(* Logix 5000 project; controller Kollmeyer_LiveDemo_TBENLX8IOL_TBIL vendor 1 type 14 code 176 rev 32.11; software revision 32.00 *)

TASK MainTask (continuous, watchdog 500 ms) : MainProgram
TASK SafetyTask (periodic, rate 20 ms, priority 10, watchdog 20 ms, safety) : SafetyProgram

MODULES
   Local : vendor 1 type 14 code 176 (Compact 0, rev 32.11)
      TBEN_L4_8IOL : ETHERNET-MODULE (Ethernet 192.168.1.7, rev 1.1, Output RPI 10 ms)
           TBEN_L4_8IOL:I.Data[0]   // Station Status Word
           TBEN_L4_8IOL:I.Data[0].0   // Module Diagnostics Available
           TBEN_L4_8IOL:I.Data[0].1   // INFO: ARGEE Project Running
           TBEN_L4_8IOL:I.Data[0].10   // Reserved
           TBEN_L4_8IOL:I.Data[0].11   // Reserved
           TBEN_L4_8IOL:I.Data[0].12   // Reserved
           TBEN_L4_8IOL:I.Data[0].13   // Reserved
           TBEN_L4_8IOL:I.Data[0].14   // Force Mode Enabled
           TBEN_L4_8IOL:I.Data[0].15   // Reserved
           TBEN_L4_8IOL:I.Data[0].2   // Reserved
           TBEN_L4_8IOL:I.Data[0].3   // Reserved
           TBEN_L4_8IOL:I.Data[0].4   // Reserved
           TBEN_L4_8IOL:I.Data[0].5   // Reserved
           TBEN_L4_8IOL:I.Data[0].6   // Reserved
           TBEN_L4_8IOL:I.Data[0].7   // Undervoltage Field Supply V2
           TBEN_L4_8IOL:I.Data[0].8   // Reserved
           TBEN_L4_8IOL:I.Data[0].9   // Undervoltage Field Supply V1
           TBEN_L4_8IOL:I.Data[100]   // IO-Link Port 7 - Input data word 1
           TBEN_L4_8IOL:I.Data[100].0   // IO-Link Port 7 - Input data word 1 (INT bit0)
           TBEN_L4_8IOL:I.Data[100].1   // IO-Link Port 7 - Input data word 1 (INT bit1)
           TBEN_L4_8IOL:I.Data[100].10   // IO-Link Port 7 - Input data word 1 (INT bit10)
           TBEN_L4_8IOL:I.Data[100].11   // IO-Link Port 7 - Input data word 1 (INT bit11)
           TBEN_L4_8IOL:I.Data[100].12   // IO-Link Port 7 - Input data word 1 (INT bit12)
           TBEN_L4_8IOL:I.Data[100].13   // IO-Link Port 7 - Input data word 1 (INT bit13)
           TBEN_L4_8IOL:I.Data[100].14   // IO-Link Port 7 - Input data word 1 (INT bit14)
           TBEN_L4_8IOL:I.Data[100].15   // IO-Link Port 7 - Input data word 1 (INT bit15)
           TBEN_L4_8IOL:I.Data[100].2   // IO-Link Port 7 - Input data word 1 (INT bit2)
           TBEN_L4_8IOL:I.Data[100].3   // IO-Link Port 7 - Input data word 1 (INT bit3)
           TBEN_L4_8IOL:I.Data[100].4   // IO-Link Port 7 - Input data word 1 (INT bit4)
           TBEN_L4_8IOL:I.Data[100].5   // IO-Link Port 7 - Input data word 1 (INT bit5)
           TBEN_L4_8IOL:I.Data[100].6   // IO-Link Port 7 - Input data word 1 (INT bit6)
           TBEN_L4_8IOL:I.Data[100].7   // IO-Link Port 7 - Input data word 1 (INT bit7)
           TBEN_L4_8IOL:I.Data[100].8   // IO-Link Port 7 - Input data word 1 (INT bit8)
           TBEN_L4_8IOL:I.Data[100].9   // IO-Link Port 7 - Input data word 1 (INT bit9)
           TBEN_L4_8IOL:I.Data[101]   // IO-Link Port 7 - Input data word 2
           TBEN_L4_8IOL:I.Data[101].0   // IO-Link Port 7 - Input data word 2 (INT bit0)
           TBEN_L4_8IOL:I.Data[101].1   // IO-Link Port 7 - Input data word 2 (INT bit1)
           TBEN_L4_8IOL:I.Data[101].10   // IO-Link Port 7 - Input data word 2 (INT bit10)
           TBEN_L4_8IOL:I.Data[101].11   // IO-Link Port 7 - Input data word 2 (INT bit11)
           TBEN_L4_8IOL:I.Data[101].12   // IO-Link Port 7 - Input data word 2 (INT bit12)
           TBEN_L4_8IOL:I.Data[101].13   // IO-Link Port 7 - Input data word 2 (INT bit13)
           TBEN_L4_8IOL:I.Data[101].14   // IO-Link Port 7 - Input data word 2 (INT bit14)
           TBEN_L4_8IOL:I.Data[101].15   // IO-Link Port 7 - Input data word 2 (INT bit15)
           TBEN_L4_8IOL:I.Data[101].2   // IO-Link Port 7 - Input data word 2 (INT bit2)
           TBEN_L4_8IOL:I.Data[101].3   // IO-Link Port 7 - Input data word 2 (INT bit3)
           TBEN_L4_8IOL:I.Data[101].4   // IO-Link Port 7 - Input data word 2 (INT bit4)
           TBEN_L4_8IOL:I.Data[101].5   // IO-Link Port 7 - Input data word 2 (INT bit5)
           TBEN_L4_8IOL:I.Data[101].6   // IO-Link Port 7 - Input data word 2 (INT bit6)
           TBEN_L4_8IOL:I.Data[101].7   // IO-Link Port 7 - Input data word 2 (INT bit7)
           TBEN_L4_8IOL:I.Data[101].8   // IO-Link Port 7 - Input data word 2 (INT bit8)
           TBEN_L4_8IOL:I.Data[101].9   // IO-Link Port 7 - Input data word 2 (INT bit9)
           TBEN_L4_8IOL:I.Data[102]   // IO-Link Port 7 - Input data word 3
           TBEN_L4_8IOL:I.Data[102].0   // IO-Link Port 7 - Input data word 3 (INT bit0)
           TBEN_L4_8IOL:I.Data[102].1   // IO-Link Port 7 - Input data word 3 (INT bit1)
           TBEN_L4_8IOL:I.Data[102].10   // IO-Link Port 7 - Input data word 3 (INT bit10)
           TBEN_L4_8IOL:I.Data[102].11   // IO-Link Port 7 - Input data word 3 (INT bit11)
           TBEN_L4_8IOL:I.Data[102].12   // IO-Link Port 7 - Input data word 3 (INT bit12)
           TBEN_L4_8IOL:I.Data[102].13   // IO-Link Port 7 - Input data word 3 (INT bit13)
           TBEN_L4_8IOL:I.Data[102].14   // IO-Link Port 7 - Input data word 3 (INT bit14)
           TBEN_L4_8IOL:I.Data[102].15   // IO-Link Port 7 - Input data word 3 (INT bit15)
           TBEN_L4_8IOL:I.Data[102].2   // IO-Link Port 7 - Input data word 3 (INT bit2)
           TBEN_L4_8IOL:I.Data[102].3   // IO-Link Port 7 - Input data word 3 (INT bit3)
           TBEN_L4_8IOL:I.Data[102].4   // IO-Link Port 7 - Input data word 3 (INT bit4)
           TBEN_L4_8IOL:I.Data[102].5   // IO-Link Port 7 - Input data word 3 (INT bit5)
           TBEN_L4_8IOL:I.Data[102].6   // IO-Link Port 7 - Input data word 3 (INT bit6)
           TBEN_L4_8IOL:I.Data[102].7   // IO-Link Port 7 - Input data word 3 (INT bit7)
           TBEN_L4_8IOL:I.Data[102].8   // IO-Link Port 7 - Input data word 3 (INT bit8)
           TBEN_L4_8IOL:I.Data[102].9   // IO-Link Port 7 - Input data word 3 (INT bit9)
           TBEN_L4_8IOL:I.Data[103]   // IO-Link Port 7 - Input data word 4
           TBEN_L4_8IOL:I.Data[103].0   // IO-Link Port 7 - Input data word 4 (INT bit0)
           TBEN_L4_8IOL:I.Data[103].1   // IO-Link Port 7 - Input data word 4 (INT bit1)
           TBEN_L4_8IOL:I.Data[103].10   // IO-Link Port 7 - Input data word 4 (INT bit10)
           TBEN_L4_8IOL:I.Data[103].11   // IO-Link Port 7 - Input data word 4 (INT bit11)
           TBEN_L4_8IOL:I.Data[103].12   // IO-Link Port 7 - Input data word 4 (INT bit12)
           TBEN_L4_8IOL:I.Data[103].13   // IO-Link Port 7 - Input data word 4 (INT bit13)
           TBEN_L4_8IOL:I.Data[103].14   // IO-Link Port 7 - Input data word 4 (INT bit14)
           TBEN_L4_8IOL:I.Data[103].15   // IO-Link Port 7 - Input data word 4 (INT bit15)
           TBEN_L4_8IOL:I.Data[103].2   // IO-Link Port 7 - Input data word 4 (INT bit2)
           TBEN_L4_8IOL:I.Data[103].3   // IO-Link Port 7 - Input data word 4 (INT bit3)
           TBEN_L4_8IOL:I.Data[103].4   // IO-Link Port 7 - Input data word 4 (INT bit4)
           TBEN_L4_8IOL:I.Data[103].5   // IO-Link Port 7 - Input data word 4 (INT bit5)
           TBEN_L4_8IOL:I.Data[103].6   // IO-Link Port 7 - Input data word 4 (INT bit6)
           TBEN_L4_8IOL:I.Data[103].7   // IO-Link Port 7 - Input data word 4 (INT bit7)
           TBEN_L4_8IOL:I.Data[103].8   // IO-Link Port 7 - Input data word 4 (INT bit8)
           TBEN_L4_8IOL:I.Data[103].9   // IO-Link Port 7 - Input data word 4 (INT bit9)
           TBEN_L4_8IOL:I.Data[104]   // IO-Link Port 7 - Input data word 5
           TBEN_L4_8IOL:I.Data[104].0   // IO-Link Port 7 - Input data word 5 (INT bit0)
           TBEN_L4_8IOL:I.Data[104].1   // IO-Link Port 7 - Input data word 5 (INT bit1)
           TBEN_L4_8IOL:I.Data[104].10   // IO-Link Port 7 - Input data word 5 (INT bit10)
           TBEN_L4_8IOL:I.Data[104].11   // IO-Link Port 7 - Input data word 5 (INT bit11)
           TBEN_L4_8IOL:I.Data[104].12   // IO-Link Port 7 - Input data word 5 (INT bit12)
           TBEN_L4_8IOL:I.Data[104].13   // IO-Link Port 7 - Input data word 5 (INT bit13)
           TBEN_L4_8IOL:I.Data[104].14   // IO-Link Port 7 - Input data word 5 (INT bit14)
           TBEN_L4_8IOL:I.Data[104].15   // IO-Link Port 7 - Input data word 5 (INT bit15)
           TBEN_L4_8IOL:I.Data[104].2   // IO-Link Port 7 - Input data word 5 (INT bit2)
           TBEN_L4_8IOL:I.Data[104].3   // IO-Link Port 7 - Input data word 5 (INT bit3)
           TBEN_L4_8IOL:I.Data[104].4   // IO-Link Port 7 - Input data word 5 (INT bit4)
           TBEN_L4_8IOL:I.Data[104].5   // IO-Link Port 7 - Input data word 5 (INT bit5)
           TBEN_L4_8IOL:I.Data[104].6   // IO-Link Port 7 - Input data word 5 (INT bit6)
           TBEN_L4_8IOL:I.Data[104].7   // IO-Link Port 7 - Input data word 5 (INT bit7)
           TBEN_L4_8IOL:I.Data[104].8   // IO-Link Port 7 - Input data word 5 (INT bit8)
           TBEN_L4_8IOL:I.Data[104].9   // IO-Link Port 7 - Input data word 5 (INT bit9)
           TBEN_L4_8IOL:I.Data[105]   // IO-Link Port 7 - Input data word 6
           TBEN_L4_8IOL:I.Data[105].0   // IO-Link Port 7 - Input data word 6 (INT bit0)
           TBEN_L4_8IOL:I.Data[105].1   // IO-Link Port 7 - Input data word 6 (INT bit1)
           TBEN_L4_8IOL:I.Data[105].10   // IO-Link Port 7 - Input data word 6 (INT bit10)
           TBEN_L4_8IOL:I.Data[105].11   // IO-Link Port 7 - Input data word 6 (INT bit11)
           TBEN_L4_8IOL:I.Data[105].12   // IO-Link Port 7 - Input data word 6 (INT bit12)
           TBEN_L4_8IOL:I.Data[105].13   // IO-Link Port 7 - Input data word 6 (INT bit13)
           TBEN_L4_8IOL:I.Data[105].14   // IO-Link Port 7 - Input data word 6 (INT bit14)
           TBEN_L4_8IOL:I.Data[105].15   // IO-Link Port 7 - Input data word 6 (INT bit15)
           TBEN_L4_8IOL:I.Data[105].2   // IO-Link Port 7 - Input data word 6 (INT bit2)
           TBEN_L4_8IOL:I.Data[105].3   // IO-Link Port 7 - Input data word 6 (INT bit3)
           TBEN_L4_8IOL:I.Data[105].4   // IO-Link Port 7 - Input data word 6 (INT bit4)
           TBEN_L4_8IOL:I.Data[105].5   // IO-Link Port 7 - Input data word 6 (INT bit5)
           TBEN_L4_8IOL:I.Data[105].6   // IO-Link Port 7 - Input data word 6 (INT bit6)
           TBEN_L4_8IOL:I.Data[105].7   // IO-Link Port 7 - Input data word 6 (INT bit7)
           TBEN_L4_8IOL:I.Data[105].8   // IO-Link Port 7 - Input data word 6 (INT bit8)
           TBEN_L4_8IOL:I.Data[105].9   // IO-Link Port 7 - Input data word 6 (INT bit9)
           TBEN_L4_8IOL:I.Data[106]   // IO-Link Port 7 - Input data word 7
           TBEN_L4_8IOL:I.Data[106].0   // IO-Link Port 7 - Input data word 7 (INT bit0)
           TBEN_L4_8IOL:I.Data[106].1   // IO-Link Port 7 - Input data word 7 (INT bit1)
           TBEN_L4_8IOL:I.Data[106].10   // IO-Link Port 7 - Input data word 7 (INT bit10)
           TBEN_L4_8IOL:I.Data[106].11   // IO-Link Port 7 - Input data word 7 (INT bit11)
           TBEN_L4_8IOL:I.Data[106].12   // IO-Link Port 7 - Input data word 7 (INT bit12)
           TBEN_L4_8IOL:I.Data[106].13   // IO-Link Port 7 - Input data word 7 (INT bit13)
           TBEN_L4_8IOL:I.Data[106].14   // IO-Link Port 7 - Input data word 7 (INT bit14)
           TBEN_L4_8IOL:I.Data[106].15   // IO-Link Port 7 - Input data word 7 (INT bit15)
           TBEN_L4_8IOL:I.Data[106].2   // IO-Link Port 7 - Input data word 7 (INT bit2)
           TBEN_L4_8IOL:I.Data[106].3   // IO-Link Port 7 - Input data word 7 (INT bit3)
           TBEN_L4_8IOL:I.Data[106].4   // IO-Link Port 7 - Input data word 7 (INT bit4)
           TBEN_L4_8IOL:I.Data[106].5   // IO-Link Port 7 - Input data word 7 (INT bit5)
           TBEN_L4_8IOL:I.Data[106].6   // IO-Link Port 7 - Input data word 7 (INT bit6)
           TBEN_L4_8IOL:I.Data[106].7   // IO-Link Port 7 - Input data word 7 (INT bit7)
           TBEN_L4_8IOL:I.Data[106].8   // IO-Link Port 7 - Input data word 7 (INT bit8)
           TBEN_L4_8IOL:I.Data[106].9   // IO-Link Port 7 - Input data word 7 (INT bit9)
           TBEN_L4_8IOL:I.Data[107]   // IO-Link Port 7 - Input data word 8
           TBEN_L4_8IOL:I.Data[107].0   // IO-Link Port 7 - Input data word 8 (INT bit0)
           TBEN_L4_8IOL:I.Data[107].1   // IO-Link Port 7 - Input data word 8 (INT bit1)
           TBEN_L4_8IOL:I.Data[107].10   // IO-Link Port 7 - Input data word 8 (INT bit10)
           TBEN_L4_8IOL:I.Data[107].11   // IO-Link Port 7 - Input data word 8 (INT bit11)
           TBEN_L4_8IOL:I.Data[107].12   // IO-Link Port 7 - Input data word 8 (INT bit12)
           TBEN_L4_8IOL:I.Data[107].13   // IO-Link Port 7 - Input data word 8 (INT bit13)
           TBEN_L4_8IOL:I.Data[107].14   // IO-Link Port 7 - Input data word 8 (INT bit14)
           TBEN_L4_8IOL:I.Data[107].15   // IO-Link Port 7 - Input data word 8 (INT bit15)
           TBEN_L4_8IOL:I.Data[107].2   // IO-Link Port 7 - Input data word 8 (INT bit2)
           TBEN_L4_8IOL:I.Data[107].3   // IO-Link Port 7 - Input data word 8 (INT bit3)
           TBEN_L4_8IOL:I.Data[107].4   // IO-Link Port 7 - Input data word 8 (INT bit4)
           TBEN_L4_8IOL:I.Data[107].5   // IO-Link Port 7 - Input data word 8 (INT bit5)
           TBEN_L4_8IOL:I.Data[107].6   // IO-Link Port 7 - Input data word 8 (INT bit6)
           TBEN_L4_8IOL:I.Data[107].7   // IO-Link Port 7 - Input data word 8 (INT bit7)
           TBEN_L4_8IOL:I.Data[107].8   // IO-Link Port 7 - Input data word 8 (INT bit8)
           TBEN_L4_8IOL:I.Data[107].9   // IO-Link Port 7 - Input data word 8 (INT bit9)
           TBEN_L4_8IOL:I.Data[108]   // IO-Link Port 7 - Input data word 9
           TBEN_L4_8IOL:I.Data[108].0   // IO-Link Port 7 - Input data word 9 (INT bit0)
           TBEN_L4_8IOL:I.Data[108].1   // IO-Link Port 7 - Input data word 9 (INT bit1)
           TBEN_L4_8IOL:I.Data[108].10   // IO-Link Port 7 - Input data word 9 (INT bit10)
           TBEN_L4_8IOL:I.Data[108].11   // IO-Link Port 7 - Input data word 9 (INT bit11)
           TBEN_L4_8IOL:I.Data[108].12   // IO-Link Port 7 - Input data word 9 (INT bit12)
           TBEN_L4_8IOL:I.Data[108].13   // IO-Link Port 7 - Input data word 9 (INT bit13)
           TBEN_L4_8IOL:I.Data[108].14   // IO-Link Port 7 - Input data word 9 (INT bit14)
           TBEN_L4_8IOL:I.Data[108].15   // IO-Link Port 7 - Input data word 9 (INT bit15)
           TBEN_L4_8IOL:I.Data[108].2   // IO-Link Port 7 - Input data word 9 (INT bit2)
           TBEN_L4_8IOL:I.Data[108].3   // IO-Link Port 7 - Input data word 9 (INT bit3)
           TBEN_L4_8IOL:I.Data[108].4   // IO-Link Port 7 - Input data word 9 (INT bit4)
           TBEN_L4_8IOL:I.Data[108].5   // IO-Link Port 7 - Input data word 9 (INT bit5)
           TBEN_L4_8IOL:I.Data[108].6   // IO-Link Port 7 - Input data word 9 (INT bit6)
           TBEN_L4_8IOL:I.Data[108].7   // IO-Link Port 7 - Input data word 9 (INT bit7)
           TBEN_L4_8IOL:I.Data[108].8   // IO-Link Port 7 - Input data word 9 (INT bit8)
           TBEN_L4_8IOL:I.Data[108].9   // IO-Link Port 7 - Input data word 9 (INT bit9)
           TBEN_L4_8IOL:I.Data[109]   // IO-Link Port 7 - Input data word 10
           TBEN_L4_8IOL:I.Data[109].0   // IO-Link Port 7 - Input data word 10 (INT bit0)
           TBEN_L4_8IOL:I.Data[109].1   // IO-Link Port 7 - Input data word 10 (INT bit1)
           TBEN_L4_8IOL:I.Data[109].10   // IO-Link Port 7 - Input data word 10 (INT bit10)
           TBEN_L4_8IOL:I.Data[109].11   // IO-Link Port 7 - Input data word 10 (INT bit11)
           TBEN_L4_8IOL:I.Data[109].12   // IO-Link Port 7 - Input data word 10 (INT bit12)
           TBEN_L4_8IOL:I.Data[109].13   // IO-Link Port 7 - Input data word 10 (INT bit13)
           TBEN_L4_8IOL:I.Data[109].14   // IO-Link Port 7 - Input data word 10 (INT bit14)
           TBEN_L4_8IOL:I.Data[109].15   // IO-Link Port 7 - Input data word 10 (INT bit15)
           TBEN_L4_8IOL:I.Data[109].2   // IO-Link Port 7 - Input data word 10 (INT bit2)
           TBEN_L4_8IOL:I.Data[109].3   // IO-Link Port 7 - Input data word 10 (INT bit3)
           TBEN_L4_8IOL:I.Data[109].4   // IO-Link Port 7 - Input data word 10 (INT bit4)
           TBEN_L4_8IOL:I.Data[109].5   // IO-Link Port 7 - Input data word 10 (INT bit5)
           TBEN_L4_8IOL:I.Data[109].6   // IO-Link Port 7 - Input data word 10 (INT bit6)
           TBEN_L4_8IOL:I.Data[109].7   // IO-Link Port 7 - Input data word 10 (INT bit7)
           TBEN_L4_8IOL:I.Data[109].8   // IO-Link Port 7 - Input data word 10 (INT bit8)
           TBEN_L4_8IOL:I.Data[109].9   // IO-Link Port 7 - Input data word 10 (INT bit9)
           TBEN_L4_8IOL:I.Data[10]   // IO-Link Port 1 - Input data word 7
           TBEN_L4_8IOL:I.Data[10].0   // IO-Link Port 1 - Input data word 7 (INT bit0)
           TBEN_L4_8IOL:I.Data[10].1   // IO-Link Port 1 - Input data word 7 (INT bit1)
           TBEN_L4_8IOL:I.Data[10].10   // IO-Link Port 1 - Input data word 7 (INT bit10)
           TBEN_L4_8IOL:I.Data[10].11   // IO-Link Port 1 - Input data word 7 (INT bit11)
           TBEN_L4_8IOL:I.Data[10].12   // IO-Link Port 1 - Input data word 7 (INT bit12)
           TBEN_L4_8IOL:I.Data[10].13   // IO-Link Port 1 - Input data word 7 (INT bit13)
           TBEN_L4_8IOL:I.Data[10].14   // IO-Link Port 1 - Input data word 7 (INT bit14)
           TBEN_L4_8IOL:I.Data[10].15   // IO-Link Port 1 - Input data word 7 (INT bit15)
           TBEN_L4_8IOL:I.Data[10].2   // IO-Link Port 1 - Input data word 7 (INT bit2)
           TBEN_L4_8IOL:I.Data[10].3   // IO-Link Port 1 - Input data word 7 (INT bit3)
           TBEN_L4_8IOL:I.Data[10].4   // IO-Link Port 1 - Input data word 7 (INT bit4)
           TBEN_L4_8IOL:I.Data[10].5   // IO-Link Port 1 - Input data word 7 (INT bit5)
           TBEN_L4_8IOL:I.Data[10].6   // IO-Link Port 1 - Input data word 7 (INT bit6)
           TBEN_L4_8IOL:I.Data[10].7   // IO-Link Port 1 - Input data word 7 (INT bit7)
           TBEN_L4_8IOL:I.Data[10].8   // IO-Link Port 1 - Input data word 7 (INT bit8)
           TBEN_L4_8IOL:I.Data[10].9   // IO-Link Port 1 - Input data word 7 (INT bit9)
           TBEN_L4_8IOL:I.Data[110]   // IO-Link Port 7 - Input data word 11
           TBEN_L4_8IOL:I.Data[110].0   // IO-Link Port 7 - Input data word 11 (INT bit0)
           TBEN_L4_8IOL:I.Data[110].1   // IO-Link Port 7 - Input data word 11 (INT bit1)
           TBEN_L4_8IOL:I.Data[110].10   // IO-Link Port 7 - Input data word 11 (INT bit10)
           TBEN_L4_8IOL:I.Data[110].11   // IO-Link Port 7 - Input data word 11 (INT bit11)
           TBEN_L4_8IOL:I.Data[110].12   // IO-Link Port 7 - Input data word 11 (INT bit12)
           TBEN_L4_8IOL:I.Data[110].13   // IO-Link Port 7 - Input data word 11 (INT bit13)
           TBEN_L4_8IOL:I.Data[110].14   // IO-Link Port 7 - Input data word 11 (INT bit14)
           TBEN_L4_8IOL:I.Data[110].15   // IO-Link Port 7 - Input data word 11 (INT bit15)
           TBEN_L4_8IOL:I.Data[110].2   // IO-Link Port 7 - Input data word 11 (INT bit2)
           TBEN_L4_8IOL:I.Data[110].3   // IO-Link Port 7 - Input data word 11 (INT bit3)
           TBEN_L4_8IOL:I.Data[110].4   // IO-Link Port 7 - Input data word 11 (INT bit4)
           TBEN_L4_8IOL:I.Data[110].5   // IO-Link Port 7 - Input data word 11 (INT bit5)
           TBEN_L4_8IOL:I.Data[110].6   // IO-Link Port 7 - Input data word 11 (INT bit6)
           TBEN_L4_8IOL:I.Data[110].7   // IO-Link Port 7 - Input data word 11 (INT bit7)
           TBEN_L4_8IOL:I.Data[110].8   // IO-Link Port 7 - Input data word 11 (INT bit8)
           TBEN_L4_8IOL:I.Data[110].9   // IO-Link Port 7 - Input data word 11 (INT bit9)
           TBEN_L4_8IOL:I.Data[111]   // IO-Link Port 7 - Input data word 12
           TBEN_L4_8IOL:I.Data[111].0   // IO-Link Port 7 - Input data word 12 (INT bit0)
           TBEN_L4_8IOL:I.Data[111].1   // IO-Link Port 7 - Input data word 12 (INT bit1)
           TBEN_L4_8IOL:I.Data[111].10   // IO-Link Port 7 - Input data word 12 (INT bit10)
           TBEN_L4_8IOL:I.Data[111].11   // IO-Link Port 7 - Input data word 12 (INT bit11)
           TBEN_L4_8IOL:I.Data[111].12   // IO-Link Port 7 - Input data word 12 (INT bit12)
           TBEN_L4_8IOL:I.Data[111].13   // IO-Link Port 7 - Input data word 12 (INT bit13)
           TBEN_L4_8IOL:I.Data[111].14   // IO-Link Port 7 - Input data word 12 (INT bit14)
           TBEN_L4_8IOL:I.Data[111].15   // IO-Link Port 7 - Input data word 12 (INT bit15)
           TBEN_L4_8IOL:I.Data[111].2   // IO-Link Port 7 - Input data word 12 (INT bit2)
           TBEN_L4_8IOL:I.Data[111].3   // IO-Link Port 7 - Input data word 12 (INT bit3)
           TBEN_L4_8IOL:I.Data[111].4   // IO-Link Port 7 - Input data word 12 (INT bit4)
           TBEN_L4_8IOL:I.Data[111].5   // IO-Link Port 7 - Input data word 12 (INT bit5)
           TBEN_L4_8IOL:I.Data[111].6   // IO-Link Port 7 - Input data word 12 (INT bit6)
           TBEN_L4_8IOL:I.Data[111].7   // IO-Link Port 7 - Input data word 12 (INT bit7)
           TBEN_L4_8IOL:I.Data[111].8   // IO-Link Port 7 - Input data word 12 (INT bit8)
           TBEN_L4_8IOL:I.Data[111].9   // IO-Link Port 7 - Input data word 12 (INT bit9)
           TBEN_L4_8IOL:I.Data[112]   // IO-Link Port 7 - Input data word 13
           TBEN_L4_8IOL:I.Data[112].0   // IO-Link Port 7 - Input data word 13 (INT bit0)
           TBEN_L4_8IOL:I.Data[112].1   // IO-Link Port 7 - Input data word 13 (INT bit1)
           TBEN_L4_8IOL:I.Data[112].10   // IO-Link Port 7 - Input data word 13 (INT bit10)
           TBEN_L4_8IOL:I.Data[112].11   // IO-Link Port 7 - Input data word 13 (INT bit11)
           TBEN_L4_8IOL:I.Data[112].12   // IO-Link Port 7 - Input data word 13 (INT bit12)
           TBEN_L4_8IOL:I.Data[112].13   // IO-Link Port 7 - Input data word 13 (INT bit13)
           TBEN_L4_8IOL:I.Data[112].14   // IO-Link Port 7 - Input data word 13 (INT bit14)
           TBEN_L4_8IOL:I.Data[112].15   // IO-Link Port 7 - Input data word 13 (INT bit15)
           TBEN_L4_8IOL:I.Data[112].2   // IO-Link Port 7 - Input data word 13 (INT bit2)
           TBEN_L4_8IOL:I.Data[112].3   // IO-Link Port 7 - Input data word 13 (INT bit3)
           TBEN_L4_8IOL:I.Data[112].4   // IO-Link Port 7 - Input data word 13 (INT bit4)
           TBEN_L4_8IOL:I.Data[112].5   // IO-Link Port 7 - Input data word 13 (INT bit5)
           TBEN_L4_8IOL:I.Data[112].6   // IO-Link Port 7 - Input data word 13 (INT bit6)
           TBEN_L4_8IOL:I.Data[112].7   // IO-Link Port 7 - Input data word 13 (INT bit7)
           TBEN_L4_8IOL:I.Data[112].8   // IO-Link Port 7 - Input data word 13 (INT bit8)
           TBEN_L4_8IOL:I.Data[112].9   // IO-Link Port 7 - Input data word 13 (INT bit9)
           TBEN_L4_8IOL:I.Data[113]   // IO-Link Port 7 - Input data word 14
           TBEN_L4_8IOL:I.Data[113].0   // IO-Link Port 7 - Input data word 14 (INT bit0)
           TBEN_L4_8IOL:I.Data[113].1   // IO-Link Port 7 - Input data word 14 (INT bit1)
           TBEN_L4_8IOL:I.Data[113].10   // IO-Link Port 7 - Input data word 14 (INT bit10)
           TBEN_L4_8IOL:I.Data[113].11   // IO-Link Port 7 - Input data word 14 (INT bit11)
           TBEN_L4_8IOL:I.Data[113].12   // IO-Link Port 7 - Input data word 14 (INT bit12)
           TBEN_L4_8IOL:I.Data[113].13   // IO-Link Port 7 - Input data word 14 (INT bit13)
           TBEN_L4_8IOL:I.Data[113].14   // IO-Link Port 7 - Input data word 14 (INT bit14)
           TBEN_L4_8IOL:I.Data[113].15   // IO-Link Port 7 - Input data word 14 (INT bit15)
           TBEN_L4_8IOL:I.Data[113].2   // IO-Link Port 7 - Input data word 14 (INT bit2)
           TBEN_L4_8IOL:I.Data[113].3   // IO-Link Port 7 - Input data word 14 (INT bit3)
           TBEN_L4_8IOL:I.Data[113].4   // IO-Link Port 7 - Input data word 14 (INT bit4)
           TBEN_L4_8IOL:I.Data[113].5   // IO-Link Port 7 - Input data word 14 (INT bit5)
           TBEN_L4_8IOL:I.Data[113].6   // IO-Link Port 7 - Input data word 14 (INT bit6)
           TBEN_L4_8IOL:I.Data[113].7   // IO-Link Port 7 - Input data word 14 (INT bit7)
           TBEN_L4_8IOL:I.Data[113].8   // IO-Link Port 7 - Input data word 14 (INT bit8)
           TBEN_L4_8IOL:I.Data[113].9   // IO-Link Port 7 - Input data word 14 (INT bit9)
           TBEN_L4_8IOL:I.Data[114]   // IO-Link Port 7 - Input data word 15
           TBEN_L4_8IOL:I.Data[114].0   // IO-Link Port 7 - Input data word 15 (INT bit0)
           TBEN_L4_8IOL:I.Data[114].1   // IO-Link Port 7 - Input data word 15 (INT bit1)
           TBEN_L4_8IOL:I.Data[114].10   // IO-Link Port 7 - Input data word 15 (INT bit10)
           TBEN_L4_8IOL:I.Data[114].11   // IO-Link Port 7 - Input data word 15 (INT bit11)
           TBEN_L4_8IOL:I.Data[114].12   // IO-Link Port 7 - Input data word 15 (INT bit12)
           TBEN_L4_8IOL:I.Data[114].13   // IO-Link Port 7 - Input data word 15 (INT bit13)
           TBEN_L4_8IOL:I.Data[114].14   // IO-Link Port 7 - Input data word 15 (INT bit14)
           TBEN_L4_8IOL:I.Data[114].15   // IO-Link Port 7 - Input data word 15 (INT bit15)
           TBEN_L4_8IOL:I.Data[114].2   // IO-Link Port 7 - Input data word 15 (INT bit2)
           TBEN_L4_8IOL:I.Data[114].3   // IO-Link Port 7 - Input data word 15 (INT bit3)
           TBEN_L4_8IOL:I.Data[114].4   // IO-Link Port 7 - Input data word 15 (INT bit4)
           TBEN_L4_8IOL:I.Data[114].5   // IO-Link Port 7 - Input data word 15 (INT bit5)
           TBEN_L4_8IOL:I.Data[114].6   // IO-Link Port 7 - Input data word 15 (INT bit6)
           TBEN_L4_8IOL:I.Data[114].7   // IO-Link Port 7 - Input data word 15 (INT bit7)
           TBEN_L4_8IOL:I.Data[114].8   // IO-Link Port 7 - Input data word 15 (INT bit8)
           TBEN_L4_8IOL:I.Data[114].9   // IO-Link Port 7 - Input data word 15 (INT bit9)
           TBEN_L4_8IOL:I.Data[115]   // IO-Link Port 8 - Input data word 0
           TBEN_L4_8IOL:I.Data[115].0   // IO-Link Port 8 - Input data word 0 (INT bit0)
           TBEN_L4_8IOL:I.Data[115].1   // IO-Link Port 8 - Input data word 0 (INT bit1)
           TBEN_L4_8IOL:I.Data[115].10   // IO-Link Port 8 - Input data word 0 (INT bit10)
           TBEN_L4_8IOL:I.Data[115].11   // IO-Link Port 8 - Input data word 0 (INT bit11)
           TBEN_L4_8IOL:I.Data[115].12   // IO-Link Port 8 - Input data word 0 (INT bit12)
           TBEN_L4_8IOL:I.Data[115].13   // IO-Link Port 8 - Input data word 0 (INT bit13)
           TBEN_L4_8IOL:I.Data[115].14   // IO-Link Port 8 - Input data word 0 (INT bit14)
           TBEN_L4_8IOL:I.Data[115].15   // IO-Link Port 8 - Input data word 0 (INT bit15)
           TBEN_L4_8IOL:I.Data[115].2   // IO-Link Port 8 - Input data word 0 (INT bit2)
           TBEN_L4_8IOL:I.Data[115].3   // IO-Link Port 8 - Input data word 0 (INT bit3)
           TBEN_L4_8IOL:I.Data[115].4   // IO-Link Port 8 - Input data word 0 (INT bit4)
           TBEN_L4_8IOL:I.Data[115].5   // IO-Link Port 8 - Input data word 0 (INT bit5)
           TBEN_L4_8IOL:I.Data[115].6   // IO-Link Port 8 - Input data word 0 (INT bit6)
           TBEN_L4_8IOL:I.Data[115].7   // IO-Link Port 8 - Input data word 0 (INT bit7)
           TBEN_L4_8IOL:I.Data[115].8   // IO-Link Port 8 - Input data word 0 (INT bit8)
           TBEN_L4_8IOL:I.Data[115].9   // IO-Link Port 8 - Input data word 0 (INT bit9)
           TBEN_L4_8IOL:I.Data[116]   // IO-Link Port 8 - Input data word 1
           TBEN_L4_8IOL:I.Data[116].0   // IO-Link Port 8 - Input data word 1 (INT bit0)
           TBEN_L4_8IOL:I.Data[116].1   // IO-Link Port 8 - Input data word 1 (INT bit1)
           TBEN_L4_8IOL:I.Data[116].10   // IO-Link Port 8 - Input data word 1 (INT bit10)
           TBEN_L4_8IOL:I.Data[116].11   // IO-Link Port 8 - Input data word 1 (INT bit11)
           TBEN_L4_8IOL:I.Data[116].12   // IO-Link Port 8 - Input data word 1 (INT bit12)
           TBEN_L4_8IOL:I.Data[116].13   // IO-Link Port 8 - Input data word 1 (INT bit13)
           TBEN_L4_8IOL:I.Data[116].14   // IO-Link Port 8 - Input data word 1 (INT bit14)
           TBEN_L4_8IOL:I.Data[116].15   // IO-Link Port 8 - Input data word 1 (INT bit15)
           TBEN_L4_8IOL:I.Data[116].2   // IO-Link Port 8 - Input data word 1 (INT bit2)
           TBEN_L4_8IOL:I.Data[116].3   // IO-Link Port 8 - Input data word 1 (INT bit3)
           TBEN_L4_8IOL:I.Data[116].4   // IO-Link Port 8 - Input data word 1 (INT bit4)
           TBEN_L4_8IOL:I.Data[116].5   // IO-Link Port 8 - Input data word 1 (INT bit5)
           TBEN_L4_8IOL:I.Data[116].6   // IO-Link Port 8 - Input data word 1 (INT bit6)
           TBEN_L4_8IOL:I.Data[116].7   // IO-Link Port 8 - Input data word 1 (INT bit7)
           TBEN_L4_8IOL:I.Data[116].8   // IO-Link Port 8 - Input data word 1 (INT bit8)
           TBEN_L4_8IOL:I.Data[116].9   // IO-Link Port 8 - Input data word 1 (INT bit9)
           TBEN_L4_8IOL:I.Data[117]   // IO-Link Port 8 - Input data word 2
           TBEN_L4_8IOL:I.Data[117].0   // IO-Link Port 8 - Input data word 2 (INT bit0)
           TBEN_L4_8IOL:I.Data[117].1   // IO-Link Port 8 - Input data word 2 (INT bit1)
           TBEN_L4_8IOL:I.Data[117].10   // IO-Link Port 8 - Input data word 2 (INT bit10)
           TBEN_L4_8IOL:I.Data[117].11   // IO-Link Port 8 - Input data word 2 (INT bit11)
           TBEN_L4_8IOL:I.Data[117].12   // IO-Link Port 8 - Input data word 2 (INT bit12)
           TBEN_L4_8IOL:I.Data[117].13   // IO-Link Port 8 - Input data word 2 (INT bit13)
           TBEN_L4_8IOL:I.Data[117].14   // IO-Link Port 8 - Input data word 2 (INT bit14)
           TBEN_L4_8IOL:I.Data[117].15   // IO-Link Port 8 - Input data word 2 (INT bit15)
           TBEN_L4_8IOL:I.Data[117].2   // IO-Link Port 8 - Input data word 2 (INT bit2)
           TBEN_L4_8IOL:I.Data[117].3   // IO-Link Port 8 - Input data word 2 (INT bit3)
           TBEN_L4_8IOL:I.Data[117].4   // IO-Link Port 8 - Input data word 2 (INT bit4)
           TBEN_L4_8IOL:I.Data[117].5   // IO-Link Port 8 - Input data word 2 (INT bit5)
           TBEN_L4_8IOL:I.Data[117].6   // IO-Link Port 8 - Input data word 2 (INT bit6)
           TBEN_L4_8IOL:I.Data[117].7   // IO-Link Port 8 - Input data word 2 (INT bit7)
           TBEN_L4_8IOL:I.Data[117].8   // IO-Link Port 8 - Input data word 2 (INT bit8)
           TBEN_L4_8IOL:I.Data[117].9   // IO-Link Port 8 - Input data word 2 (INT bit9)
           TBEN_L4_8IOL:I.Data[118]   // IO-Link Port 8 - Input data word 3
           TBEN_L4_8IOL:I.Data[118].0   // IO-Link Port 8 - Input data word 3 (INT bit0)
           TBEN_L4_8IOL:I.Data[118].1   // IO-Link Port 8 - Input data word 3 (INT bit1)
           TBEN_L4_8IOL:I.Data[118].10   // IO-Link Port 8 - Input data word 3 (INT bit10)
           TBEN_L4_8IOL:I.Data[118].11   // IO-Link Port 8 - Input data word 3 (INT bit11)
           TBEN_L4_8IOL:I.Data[118].12   // IO-Link Port 8 - Input data word 3 (INT bit12)
           TBEN_L4_8IOL:I.Data[118].13   // IO-Link Port 8 - Input data word 3 (INT bit13)
           TBEN_L4_8IOL:I.Data[118].14   // IO-Link Port 8 - Input data word 3 (INT bit14)
           TBEN_L4_8IOL:I.Data[118].15   // IO-Link Port 8 - Input data word 3 (INT bit15)
           TBEN_L4_8IOL:I.Data[118].2   // IO-Link Port 8 - Input data word 3 (INT bit2)
           TBEN_L4_8IOL:I.Data[118].3   // IO-Link Port 8 - Input data word 3 (INT bit3)
           TBEN_L4_8IOL:I.Data[118].4   // IO-Link Port 8 - Input data word 3 (INT bit4)
           TBEN_L4_8IOL:I.Data[118].5   // IO-Link Port 8 - Input data word 3 (INT bit5)
           TBEN_L4_8IOL:I.Data[118].6   // IO-Link Port 8 - Input data word 3 (INT bit6)
           TBEN_L4_8IOL:I.Data[118].7   // IO-Link Port 8 - Input data word 3 (INT bit7)
           TBEN_L4_8IOL:I.Data[118].8   // IO-Link Port 8 - Input data word 3 (INT bit8)
           TBEN_L4_8IOL:I.Data[118].9   // IO-Link Port 8 - Input data word 3 (INT bit9)
           TBEN_L4_8IOL:I.Data[119]   // IO-Link Port 8 - Input data word 4
           TBEN_L4_8IOL:I.Data[119].0   // IO-Link Port 8 - Input data word 4 (INT bit0)
           TBEN_L4_8IOL:I.Data[119].1   // IO-Link Port 8 - Input data word 4 (INT bit1)
           TBEN_L4_8IOL:I.Data[119].10   // IO-Link Port 8 - Input data word 4 (INT bit10)
           TBEN_L4_8IOL:I.Data[119].11   // IO-Link Port 8 - Input data word 4 (INT bit11)
           TBEN_L4_8IOL:I.Data[119].12   // IO-Link Port 8 - Input data word 4 (INT bit12)
           TBEN_L4_8IOL:I.Data[119].13   // IO-Link Port 8 - Input data word 4 (INT bit13)
           TBEN_L4_8IOL:I.Data[119].14   // IO-Link Port 8 - Input data word 4 (INT bit14)
           TBEN_L4_8IOL:I.Data[119].15   // IO-Link Port 8 - Input data word 4 (INT bit15)
           TBEN_L4_8IOL:I.Data[119].2   // IO-Link Port 8 - Input data word 4 (INT bit2)
           TBEN_L4_8IOL:I.Data[119].3   // IO-Link Port 8 - Input data word 4 (INT bit3)
           TBEN_L4_8IOL:I.Data[119].4   // IO-Link Port 8 - Input data word 4 (INT bit4)
           TBEN_L4_8IOL:I.Data[119].5   // IO-Link Port 8 - Input data word 4 (INT bit5)
           TBEN_L4_8IOL:I.Data[119].6   // IO-Link Port 8 - Input data word 4 (INT bit6)
           TBEN_L4_8IOL:I.Data[119].7   // IO-Link Port 8 - Input data word 4 (INT bit7)
           TBEN_L4_8IOL:I.Data[119].8   // IO-Link Port 8 - Input data word 4 (INT bit8)
           TBEN_L4_8IOL:I.Data[119].9   // IO-Link Port 8 - Input data word 4 (INT bit9)
           TBEN_L4_8IOL:I.Data[11]   // IO-Link Port 1 - Input data word 8
           TBEN_L4_8IOL:I.Data[11].0   // IO-Link Port 1 - Input data word 8 (INT bit0)
           TBEN_L4_8IOL:I.Data[11].1   // IO-Link Port 1 - Input data word 8 (INT bit1)
           TBEN_L4_8IOL:I.Data[11].10   // IO-Link Port 1 - Input data word 8 (INT bit10)
           TBEN_L4_8IOL:I.Data[11].11   // IO-Link Port 1 - Input data word 8 (INT bit11)
           TBEN_L4_8IOL:I.Data[11].12   // IO-Link Port 1 - Input data word 8 (INT bit12)
           TBEN_L4_8IOL:I.Data[11].13   // IO-Link Port 1 - Input data word 8 (INT bit13)
           TBEN_L4_8IOL:I.Data[11].14   // IO-Link Port 1 - Input data word 8 (INT bit14)
           TBEN_L4_8IOL:I.Data[11].15   // IO-Link Port 1 - Input data word 8 (INT bit15)
           TBEN_L4_8IOL:I.Data[11].2   // IO-Link Port 1 - Input data word 8 (INT bit2)
           TBEN_L4_8IOL:I.Data[11].3   // IO-Link Port 1 - Input data word 8 (INT bit3)
           TBEN_L4_8IOL:I.Data[11].4   // IO-Link Port 1 - Input data word 8 (INT bit4)
           TBEN_L4_8IOL:I.Data[11].5   // IO-Link Port 1 - Input data word 8 (INT bit5)
           TBEN_L4_8IOL:I.Data[11].6   // IO-Link Port 1 - Input data word 8 (INT bit6)
           TBEN_L4_8IOL:I.Data[11].7   // IO-Link Port 1 - Input data word 8 (INT bit7)
           TBEN_L4_8IOL:I.Data[11].8   // IO-Link Port 1 - Input data word 8 (INT bit8)
           TBEN_L4_8IOL:I.Data[11].9   // IO-Link Port 1 - Input data word 8 (INT bit9)
           TBEN_L4_8IOL:I.Data[120]   // IO-Link Port 8 - Input data word 5
           TBEN_L4_8IOL:I.Data[120].0   // IO-Link Port 8 - Input data word 5 (INT bit0)
           TBEN_L4_8IOL:I.Data[120].1   // IO-Link Port 8 - Input data word 5 (INT bit1)
           TBEN_L4_8IOL:I.Data[120].10   // IO-Link Port 8 - Input data word 5 (INT bit10)
           TBEN_L4_8IOL:I.Data[120].11   // IO-Link Port 8 - Input data word 5 (INT bit11)
           TBEN_L4_8IOL:I.Data[120].12   // IO-Link Port 8 - Input data word 5 (INT bit12)
           TBEN_L4_8IOL:I.Data[120].13   // IO-Link Port 8 - Input data word 5 (INT bit13)
           TBEN_L4_8IOL:I.Data[120].14   // IO-Link Port 8 - Input data word 5 (INT bit14)
           TBEN_L4_8IOL:I.Data[120].15   // IO-Link Port 8 - Input data word 5 (INT bit15)
           TBEN_L4_8IOL:I.Data[120].2   // IO-Link Port 8 - Input data word 5 (INT bit2)
           TBEN_L4_8IOL:I.Data[120].3   // IO-Link Port 8 - Input data word 5 (INT bit3)
           TBEN_L4_8IOL:I.Data[120].4   // IO-Link Port 8 - Input data word 5 (INT bit4)
           TBEN_L4_8IOL:I.Data[120].5   // IO-Link Port 8 - Input data word 5 (INT bit5)
           TBEN_L4_8IOL:I.Data[120].6   // IO-Link Port 8 - Input data word 5 (INT bit6)
           TBEN_L4_8IOL:I.Data[120].7   // IO-Link Port 8 - Input data word 5 (INT bit7)
           TBEN_L4_8IOL:I.Data[120].8   // IO-Link Port 8 - Input data word 5 (INT bit8)
           TBEN_L4_8IOL:I.Data[120].9   // IO-Link Port 8 - Input data word 5 (INT bit9)
           TBEN_L4_8IOL:I.Data[121]   // IO-Link Port 8 - Input data word 6
           TBEN_L4_8IOL:I.Data[121].0   // IO-Link Port 8 - Input data word 6 (INT bit0)
           TBEN_L4_8IOL:I.Data[121].1   // IO-Link Port 8 - Input data word 6 (INT bit1)
           TBEN_L4_8IOL:I.Data[121].10   // IO-Link Port 8 - Input data word 6 (INT bit10)
           TBEN_L4_8IOL:I.Data[121].11   // IO-Link Port 8 - Input data word 6 (INT bit11)
           TBEN_L4_8IOL:I.Data[121].12   // IO-Link Port 8 - Input data word 6 (INT bit12)
           TBEN_L4_8IOL:I.Data[121].13   // IO-Link Port 8 - Input data word 6 (INT bit13)
           TBEN_L4_8IOL:I.Data[121].14   // IO-Link Port 8 - Input data word 6 (INT bit14)
           TBEN_L4_8IOL:I.Data[121].15   // IO-Link Port 8 - Input data word 6 (INT bit15)
           TBEN_L4_8IOL:I.Data[121].2   // IO-Link Port 8 - Input data word 6 (INT bit2)
           TBEN_L4_8IOL:I.Data[121].3   // IO-Link Port 8 - Input data word 6 (INT bit3)
           TBEN_L4_8IOL:I.Data[121].4   // IO-Link Port 8 - Input data word 6 (INT bit4)
           TBEN_L4_8IOL:I.Data[121].5   // IO-Link Port 8 - Input data word 6 (INT bit5)
           TBEN_L4_8IOL:I.Data[121].6   // IO-Link Port 8 - Input data word 6 (INT bit6)
           TBEN_L4_8IOL:I.Data[121].7   // IO-Link Port 8 - Input data word 6 (INT bit7)
           TBEN_L4_8IOL:I.Data[121].8   // IO-Link Port 8 - Input data word 6 (INT bit8)
           TBEN_L4_8IOL:I.Data[121].9   // IO-Link Port 8 - Input data word 6 (INT bit9)
           TBEN_L4_8IOL:I.Data[122]   // IO-Link Port 8 - Input data word 7
           TBEN_L4_8IOL:I.Data[122].0   // IO-Link Port 8 - Input data word 7 (INT bit0)
           TBEN_L4_8IOL:I.Data[122].1   // IO-Link Port 8 - Input data word 7 (INT bit1)
           TBEN_L4_8IOL:I.Data[122].10   // IO-Link Port 8 - Input data word 7 (INT bit10)
           TBEN_L4_8IOL:I.Data[122].11   // IO-Link Port 8 - Input data word 7 (INT bit11)
           TBEN_L4_8IOL:I.Data[122].12   // IO-Link Port 8 - Input data word 7 (INT bit12)
           TBEN_L4_8IOL:I.Data[122].13   // IO-Link Port 8 - Input data word 7 (INT bit13)
           TBEN_L4_8IOL:I.Data[122].14   // IO-Link Port 8 - Input data word 7 (INT bit14)
           TBEN_L4_8IOL:I.Data[122].15   // IO-Link Port 8 - Input data word 7 (INT bit15)
           TBEN_L4_8IOL:I.Data[122].2   // IO-Link Port 8 - Input data word 7 (INT bit2)
           TBEN_L4_8IOL:I.Data[122].3   // IO-Link Port 8 - Input data word 7 (INT bit3)
           TBEN_L4_8IOL:I.Data[122].4   // IO-Link Port 8 - Input data word 7 (INT bit4)
           TBEN_L4_8IOL:I.Data[122].5   // IO-Link Port 8 - Input data word 7 (INT bit5)
           TBEN_L4_8IOL:I.Data[122].6   // IO-Link Port 8 - Input data word 7 (INT bit6)
           TBEN_L4_8IOL:I.Data[122].7   // IO-Link Port 8 - Input data word 7 (INT bit7)
           TBEN_L4_8IOL:I.Data[122].8   // IO-Link Port 8 - Input data word 7 (INT bit8)
           TBEN_L4_8IOL:I.Data[122].9   // IO-Link Port 8 - Input data word 7 (INT bit9)
           TBEN_L4_8IOL:I.Data[123]   // IO-Link Port 8 - Input data word 8
           TBEN_L4_8IOL:I.Data[123].0   // IO-Link Port 8 - Input data word 8 (INT bit0)
           TBEN_L4_8IOL:I.Data[123].1   // IO-Link Port 8 - Input data word 8 (INT bit1)
           TBEN_L4_8IOL:I.Data[123].10   // IO-Link Port 8 - Input data word 8 (INT bit10)
           TBEN_L4_8IOL:I.Data[123].11   // IO-Link Port 8 - Input data word 8 (INT bit11)
           TBEN_L4_8IOL:I.Data[123].12   // IO-Link Port 8 - Input data word 8 (INT bit12)
           TBEN_L4_8IOL:I.Data[123].13   // IO-Link Port 8 - Input data word 8 (INT bit13)
           TBEN_L4_8IOL:I.Data[123].14   // IO-Link Port 8 - Input data word 8 (INT bit14)
           TBEN_L4_8IOL:I.Data[123].15   // IO-Link Port 8 - Input data word 8 (INT bit15)
           TBEN_L4_8IOL:I.Data[123].2   // IO-Link Port 8 - Input data word 8 (INT bit2)
           TBEN_L4_8IOL:I.Data[123].3   // IO-Link Port 8 - Input data word 8 (INT bit3)
           TBEN_L4_8IOL:I.Data[123].4   // IO-Link Port 8 - Input data word 8 (INT bit4)
           TBEN_L4_8IOL:I.Data[123].5   // IO-Link Port 8 - Input data word 8 (INT bit5)
           TBEN_L4_8IOL:I.Data[123].6   // IO-Link Port 8 - Input data word 8 (INT bit6)
           TBEN_L4_8IOL:I.Data[123].7   // IO-Link Port 8 - Input data word 8 (INT bit7)
           TBEN_L4_8IOL:I.Data[123].8   // IO-Link Port 8 - Input data word 8 (INT bit8)
           TBEN_L4_8IOL:I.Data[123].9   // IO-Link Port 8 - Input data word 8 (INT bit9)
           TBEN_L4_8IOL:I.Data[124]   // IO-Link Port 8 - Input data word 9
           TBEN_L4_8IOL:I.Data[124].0   // IO-Link Port 8 - Input data word 9 (INT bit0)
           TBEN_L4_8IOL:I.Data[124].1   // IO-Link Port 8 - Input data word 9 (INT bit1)
           TBEN_L4_8IOL:I.Data[124].10   // IO-Link Port 8 - Input data word 9 (INT bit10)
           TBEN_L4_8IOL:I.Data[124].11   // IO-Link Port 8 - Input data word 9 (INT bit11)
           TBEN_L4_8IOL:I.Data[124].12   // IO-Link Port 8 - Input data word 9 (INT bit12)
           TBEN_L4_8IOL:I.Data[124].13   // IO-Link Port 8 - Input data word 9 (INT bit13)
           TBEN_L4_8IOL:I.Data[124].14   // IO-Link Port 8 - Input data word 9 (INT bit14)
           TBEN_L4_8IOL:I.Data[124].15   // IO-Link Port 8 - Input data word 9 (INT bit15)
           TBEN_L4_8IOL:I.Data[124].2   // IO-Link Port 8 - Input data word 9 (INT bit2)
           TBEN_L4_8IOL:I.Data[124].3   // IO-Link Port 8 - Input data word 9 (INT bit3)
           TBEN_L4_8IOL:I.Data[124].4   // IO-Link Port 8 - Input data word 9 (INT bit4)
           TBEN_L4_8IOL:I.Data[124].5   // IO-Link Port 8 - Input data word 9 (INT bit5)
           TBEN_L4_8IOL:I.Data[124].6   // IO-Link Port 8 - Input data word 9 (INT bit6)
           TBEN_L4_8IOL:I.Data[124].7   // IO-Link Port 8 - Input data word 9 (INT bit7)
           TBEN_L4_8IOL:I.Data[124].8   // IO-Link Port 8 - Input data word 9 (INT bit8)
           TBEN_L4_8IOL:I.Data[124].9   // IO-Link Port 8 - Input data word 9 (INT bit9)
           TBEN_L4_8IOL:I.Data[125]   // IO-Link Port 8 - Input data word 10
           TBEN_L4_8IOL:I.Data[125].0   // IO-Link Port 8 - Input data word 10 (INT bit0)
           TBEN_L4_8IOL:I.Data[125].1   // IO-Link Port 8 - Input data word 10 (INT bit1)
           TBEN_L4_8IOL:I.Data[125].10   // IO-Link Port 8 - Input data word 10 (INT bit10)
           TBEN_L4_8IOL:I.Data[125].11   // IO-Link Port 8 - Input data word 10 (INT bit11)
           TBEN_L4_8IOL:I.Data[125].12   // IO-Link Port 8 - Input data word 10 (INT bit12)
           TBEN_L4_8IOL:I.Data[125].13   // IO-Link Port 8 - Input data word 10 (INT bit13)
           TBEN_L4_8IOL:I.Data[125].14   // IO-Link Port 8 - Input data word 10 (INT bit14)
           TBEN_L4_8IOL:I.Data[125].15   // IO-Link Port 8 - Input data word 10 (INT bit15)
           TBEN_L4_8IOL:I.Data[125].2   // IO-Link Port 8 - Input data word 10 (INT bit2)
           TBEN_L4_8IOL:I.Data[125].3   // IO-Link Port 8 - Input data word 10 (INT bit3)
           TBEN_L4_8IOL:I.Data[125].4   // IO-Link Port 8 - Input data word 10 (INT bit4)
           TBEN_L4_8IOL:I.Data[125].5   // IO-Link Port 8 - Input data word 10 (INT bit5)
           TBEN_L4_8IOL:I.Data[125].6   // IO-Link Port 8 - Input data word 10 (INT bit6)
           TBEN_L4_8IOL:I.Data[125].7   // IO-Link Port 8 - Input data word 10 (INT bit7)
           TBEN_L4_8IOL:I.Data[125].8   // IO-Link Port 8 - Input data word 10 (INT bit8)
           TBEN_L4_8IOL:I.Data[125].9   // IO-Link Port 8 - Input data word 10 (INT bit9)
           TBEN_L4_8IOL:I.Data[126]   // IO-Link Port 8 - Input data word 11
           TBEN_L4_8IOL:I.Data[126].0   // IO-Link Port 8 - Input data word 11 (INT bit0)
           TBEN_L4_8IOL:I.Data[126].1   // IO-Link Port 8 - Input data word 11 (INT bit1)
           TBEN_L4_8IOL:I.Data[126].10   // IO-Link Port 8 - Input data word 11 (INT bit10)
           TBEN_L4_8IOL:I.Data[126].11   // IO-Link Port 8 - Input data word 11 (INT bit11)
           TBEN_L4_8IOL:I.Data[126].12   // IO-Link Port 8 - Input data word 11 (INT bit12)
           TBEN_L4_8IOL:I.Data[126].13   // IO-Link Port 8 - Input data word 11 (INT bit13)
           TBEN_L4_8IOL:I.Data[126].14   // IO-Link Port 8 - Input data word 11 (INT bit14)
           TBEN_L4_8IOL:I.Data[126].15   // IO-Link Port 8 - Input data word 11 (INT bit15)
           TBEN_L4_8IOL:I.Data[126].2   // IO-Link Port 8 - Input data word 11 (INT bit2)
           TBEN_L4_8IOL:I.Data[126].3   // IO-Link Port 8 - Input data word 11 (INT bit3)
           TBEN_L4_8IOL:I.Data[126].4   // IO-Link Port 8 - Input data word 11 (INT bit4)
           TBEN_L4_8IOL:I.Data[126].5   // IO-Link Port 8 - Input data word 11 (INT bit5)
           TBEN_L4_8IOL:I.Data[126].6   // IO-Link Port 8 - Input data word 11 (INT bit6)
           TBEN_L4_8IOL:I.Data[126].7   // IO-Link Port 8 - Input data word 11 (INT bit7)
           TBEN_L4_8IOL:I.Data[126].8   // IO-Link Port 8 - Input data word 11 (INT bit8)
           TBEN_L4_8IOL:I.Data[126].9   // IO-Link Port 8 - Input data word 11 (INT bit9)
           TBEN_L4_8IOL:I.Data[127]   // IO-Link Port 8 - Input data word 12
           TBEN_L4_8IOL:I.Data[127].0   // IO-Link Port 8 - Input data word 12 (INT bit0)
           TBEN_L4_8IOL:I.Data[127].1   // IO-Link Port 8 - Input data word 12 (INT bit1)
           TBEN_L4_8IOL:I.Data[127].10   // IO-Link Port 8 - Input data word 12 (INT bit10)
           TBEN_L4_8IOL:I.Data[127].11   // IO-Link Port 8 - Input data word 12 (INT bit11)
           TBEN_L4_8IOL:I.Data[127].12   // IO-Link Port 8 - Input data word 12 (INT bit12)
           TBEN_L4_8IOL:I.Data[127].13   // IO-Link Port 8 - Input data word 12 (INT bit13)
           TBEN_L4_8IOL:I.Data[127].14   // IO-Link Port 8 - Input data word 12 (INT bit14)
           TBEN_L4_8IOL:I.Data[127].15   // IO-Link Port 8 - Input data word 12 (INT bit15)
           TBEN_L4_8IOL:I.Data[127].2   // IO-Link Port 8 - Input data word 12 (INT bit2)
           TBEN_L4_8IOL:I.Data[127].3   // IO-Link Port 8 - Input data word 12 (INT bit3)
           TBEN_L4_8IOL:I.Data[127].4   // IO-Link Port 8 - Input data word 12 (INT bit4)
           TBEN_L4_8IOL:I.Data[127].5   // IO-Link Port 8 - Input data word 12 (INT bit5)
           TBEN_L4_8IOL:I.Data[127].6   // IO-Link Port 8 - Input data word 12 (INT bit6)
           TBEN_L4_8IOL:I.Data[127].7   // IO-Link Port 8 - Input data word 12 (INT bit7)
           TBEN_L4_8IOL:I.Data[127].8   // IO-Link Port 8 - Input data word 12 (INT bit8)
           TBEN_L4_8IOL:I.Data[127].9   // IO-Link Port 8 - Input data word 12 (INT bit9)
           TBEN_L4_8IOL:I.Data[128]   // IO-Link Port 8 - Input data word 13
           TBEN_L4_8IOL:I.Data[128].0   // IO-Link Port 8 - Input data word 13 (INT bit0)
           TBEN_L4_8IOL:I.Data[128].1   // IO-Link Port 8 - Input data word 13 (INT bit1)
           TBEN_L4_8IOL:I.Data[128].10   // IO-Link Port 8 - Input data word 13 (INT bit10)
           TBEN_L4_8IOL:I.Data[128].11   // IO-Link Port 8 - Input data word 13 (INT bit11)
           TBEN_L4_8IOL:I.Data[128].12   // IO-Link Port 8 - Input data word 13 (INT bit12)
           TBEN_L4_8IOL:I.Data[128].13   // IO-Link Port 8 - Input data word 13 (INT bit13)
           TBEN_L4_8IOL:I.Data[128].14   // IO-Link Port 8 - Input data word 13 (INT bit14)
           TBEN_L4_8IOL:I.Data[128].15   // IO-Link Port 8 - Input data word 13 (INT bit15)
           TBEN_L4_8IOL:I.Data[128].2   // IO-Link Port 8 - Input data word 13 (INT bit2)
           TBEN_L4_8IOL:I.Data[128].3   // IO-Link Port 8 - Input data word 13 (INT bit3)
           TBEN_L4_8IOL:I.Data[128].4   // IO-Link Port 8 - Input data word 13 (INT bit4)
           TBEN_L4_8IOL:I.Data[128].5   // IO-Link Port 8 - Input data word 13 (INT bit5)
           TBEN_L4_8IOL:I.Data[128].6   // IO-Link Port 8 - Input data word 13 (INT bit6)
           TBEN_L4_8IOL:I.Data[128].7   // IO-Link Port 8 - Input data word 13 (INT bit7)
           TBEN_L4_8IOL:I.Data[128].8   // IO-Link Port 8 - Input data word 13 (INT bit8)
           TBEN_L4_8IOL:I.Data[128].9   // IO-Link Port 8 - Input data word 13 (INT bit9)
           TBEN_L4_8IOL:I.Data[129]   // IO-Link Port 8 - Input data word 14
           TBEN_L4_8IOL:I.Data[129].0   // IO-Link Port 8 - Input data word 14 (INT bit0)
           TBEN_L4_8IOL:I.Data[129].1   // IO-Link Port 8 - Input data word 14 (INT bit1)
           TBEN_L4_8IOL:I.Data[129].10   // IO-Link Port 8 - Input data word 14 (INT bit10)
           TBEN_L4_8IOL:I.Data[129].11   // IO-Link Port 8 - Input data word 14 (INT bit11)
           TBEN_L4_8IOL:I.Data[129].12   // IO-Link Port 8 - Input data word 14 (INT bit12)
           TBEN_L4_8IOL:I.Data[129].13   // IO-Link Port 8 - Input data word 14 (INT bit13)
           TBEN_L4_8IOL:I.Data[129].14   // IO-Link Port 8 - Input data word 14 (INT bit14)
           TBEN_L4_8IOL:I.Data[129].15   // IO-Link Port 8 - Input data word 14 (INT bit15)
           TBEN_L4_8IOL:I.Data[129].2   // IO-Link Port 8 - Input data word 14 (INT bit2)
           TBEN_L4_8IOL:I.Data[129].3   // IO-Link Port 8 - Input data word 14 (INT bit3)
           TBEN_L4_8IOL:I.Data[129].4   // IO-Link Port 8 - Input data word 14 (INT bit4)
           TBEN_L4_8IOL:I.Data[129].5   // IO-Link Port 8 - Input data word 14 (INT bit5)
           TBEN_L4_8IOL:I.Data[129].6   // IO-Link Port 8 - Input data word 14 (INT bit6)
           TBEN_L4_8IOL:I.Data[129].7   // IO-Link Port 8 - Input data word 14 (INT bit7)
           TBEN_L4_8IOL:I.Data[129].8   // IO-Link Port 8 - Input data word 14 (INT bit8)
           TBEN_L4_8IOL:I.Data[129].9   // IO-Link Port 8 - Input data word 14 (INT bit9)
           TBEN_L4_8IOL:I.Data[12]   // IO-Link Port 1 - Input data word 9
           TBEN_L4_8IOL:I.Data[12].0   // IO-Link Port 1 - Input data word 9 (INT bit0)
           TBEN_L4_8IOL:I.Data[12].1   // IO-Link Port 1 - Input data word 9 (INT bit1)
           TBEN_L4_8IOL:I.Data[12].10   // IO-Link Port 1 - Input data word 9 (INT bit10)
           TBEN_L4_8IOL:I.Data[12].11   // IO-Link Port 1 - Input data word 9 (INT bit11)
           TBEN_L4_8IOL:I.Data[12].12   // IO-Link Port 1 - Input data word 9 (INT bit12)
           TBEN_L4_8IOL:I.Data[12].13   // IO-Link Port 1 - Input data word 9 (INT bit13)
           TBEN_L4_8IOL:I.Data[12].14   // IO-Link Port 1 - Input data word 9 (INT bit14)
           TBEN_L4_8IOL:I.Data[12].15   // IO-Link Port 1 - Input data word 9 (INT bit15)
           TBEN_L4_8IOL:I.Data[12].2   // IO-Link Port 1 - Input data word 9 (INT bit2)
           TBEN_L4_8IOL:I.Data[12].3   // IO-Link Port 1 - Input data word 9 (INT bit3)
           TBEN_L4_8IOL:I.Data[12].4   // IO-Link Port 1 - Input data word 9 (INT bit4)
           TBEN_L4_8IOL:I.Data[12].5   // IO-Link Port 1 - Input data word 9 (INT bit5)
           TBEN_L4_8IOL:I.Data[12].6   // IO-Link Port 1 - Input data word 9 (INT bit6)
           TBEN_L4_8IOL:I.Data[12].7   // IO-Link Port 1 - Input data word 9 (INT bit7)
           TBEN_L4_8IOL:I.Data[12].8   // IO-Link Port 1 - Input data word 9 (INT bit8)
           TBEN_L4_8IOL:I.Data[12].9   // IO-Link Port 1 - Input data word 9 (INT bit9)
           TBEN_L4_8IOL:I.Data[130]   // IO-Link Port 8 - Input data word 15
           TBEN_L4_8IOL:I.Data[130].0   // IO-Link Port 8 - Input data word 15 (INT bit0)
           TBEN_L4_8IOL:I.Data[130].1   // IO-Link Port 8 - Input data word 15 (INT bit1)
           TBEN_L4_8IOL:I.Data[130].10   // IO-Link Port 8 - Input data word 15 (INT bit10)
           TBEN_L4_8IOL:I.Data[130].11   // IO-Link Port 8 - Input data word 15 (INT bit11)
           TBEN_L4_8IOL:I.Data[130].12   // IO-Link Port 8 - Input data word 15 (INT bit12)
           TBEN_L4_8IOL:I.Data[130].13   // IO-Link Port 8 - Input data word 15 (INT bit13)
           TBEN_L4_8IOL:I.Data[130].14   // IO-Link Port 8 - Input data word 15 (INT bit14)
           TBEN_L4_8IOL:I.Data[130].15   // IO-Link Port 8 - Input data word 15 (INT bit15)
           TBEN_L4_8IOL:I.Data[130].2   // IO-Link Port 8 - Input data word 15 (INT bit2)
           TBEN_L4_8IOL:I.Data[130].3   // IO-Link Port 8 - Input data word 15 (INT bit3)
           TBEN_L4_8IOL:I.Data[130].4   // IO-Link Port 8 - Input data word 15 (INT bit4)
           TBEN_L4_8IOL:I.Data[130].5   // IO-Link Port 8 - Input data word 15 (INT bit5)
           TBEN_L4_8IOL:I.Data[130].6   // IO-Link Port 8 - Input data word 15 (INT bit6)
           TBEN_L4_8IOL:I.Data[130].7   // IO-Link Port 8 - Input data word 15 (INT bit7)
           TBEN_L4_8IOL:I.Data[130].8   // IO-Link Port 8 - Input data word 15 (INT bit8)
           TBEN_L4_8IOL:I.Data[130].9   // IO-Link Port 8 - Input data word 15 (INT bit9)
           TBEN_L4_8IOL:I.Data[131]   // Overcurrent VAUX1 Pin1 C0 (Ch0/1), Overcurrent VAUX1 Pin1 C1 (Ch2/3), Overcurrent VAUX1 Pin1 C2 (Ch4/5), Overcurrent VAUX1 Pin1 C3 (Ch6/7), Overcurrent VAUX1 Pin1 C4 (Ch8), Overcurrent VAUX1 Pin1 C5 (Ch10), Overcurrent VAUX1 Pin1 C6 (Ch12), Overcurrent VAUX1 Pin1 C7 (Ch14), Overcurrent VAUX2 Pin2 C4 (Ch9), Overcurrent VAUX2 Pin2 C5 (Ch11), Overcurrent VAUX2 Pin2 C6 (Ch13), Overcurrent VAUX2 Pin2 C7 (Ch15)
           TBEN_L4_8IOL:I.Data[131].0   // Overcurrent VAUX1 Pin1 C0 (Ch0/1) (ENUM bit0): 0=-, 1=active
           TBEN_L4_8IOL:I.Data[131].1   // Overcurrent VAUX1 Pin1 C1 (Ch2/3) (ENUM bit0): 0=-, 1=active
           TBEN_L4_8IOL:I.Data[131].10   // Reserved
           TBEN_L4_8IOL:I.Data[131].11   // Reserved
           TBEN_L4_8IOL:I.Data[131].12   // Overcurrent VAUX2 Pin2 C4 (Ch9) (ENUM bit0): 0=-, 1=active
           TBEN_L4_8IOL:I.Data[131].13   // Overcurrent VAUX2 Pin2 C5 (Ch11) (ENUM bit0): 0=-, 1=active
           TBEN_L4_8IOL:I.Data[131].14   // Overcurrent VAUX2 Pin2 C6 (Ch13) (ENUM bit0): 0=-, 1=active
           TBEN_L4_8IOL:I.Data[131].15   // Overcurrent VAUX2 Pin2 C7 (Ch15) (ENUM bit0): 0=-, 1=active
           TBEN_L4_8IOL:I.Data[131].2   // Overcurrent VAUX1 Pin1 C2 (Ch4/5) (ENUM bit0): 0=-, 1=active
           TBEN_L4_8IOL:I.Data[131].3   // Overcurrent VAUX1 Pin1 C3 (Ch6/7) (ENUM bit0): 0=-, 1=active
           TBEN_L4_8IOL:I.Data[131].4   // Overcurrent VAUX1 Pin1 C4 (Ch8) (ENUM bit0): 0=-, 1=active
           TBEN_L4_8IOL:I.Data[131].5   // Overcurrent VAUX1 Pin1 C5 (Ch10) (ENUM bit0): 0=-, 1=active
           TBEN_L4_8IOL:I.Data[131].6   // Overcurrent VAUX1 Pin1 C6 (Ch12) (ENUM bit0): 0=-, 1=active
           TBEN_L4_8IOL:I.Data[131].7   // Overcurrent VAUX1 Pin1 C7 (Ch14) (ENUM bit0): 0=-, 1=active
           TBEN_L4_8IOL:I.Data[131].8   // Reserved
           TBEN_L4_8IOL:I.Data[131].9   // Reserved
           TBEN_L4_8IOL:I.Data[132]   // DXP channel 1 - Output overcurrent, DXP channel 3 - Output overcurrent, DXP channel 5 - Output overcurrent, DXP channel 7 - Output overcurrent
           TBEN_L4_8IOL:I.Data[132].0   // Reserved
           TBEN_L4_8IOL:I.Data[132].1   // DXP channel 1 - Output overcurrent (ENUM bit0): 0=-, 1=active
           TBEN_L4_8IOL:I.Data[132].10   // Reserved
           TBEN_L4_8IOL:I.Data[132].11   // Reserved
           TBEN_L4_8IOL:I.Data[132].12   // Reserved
           TBEN_L4_8IOL:I.Data[132].13   // Reserved
           TBEN_L4_8IOL:I.Data[132].14   // Reserved
           TBEN_L4_8IOL:I.Data[132].15   // Reserved
           TBEN_L4_8IOL:I.Data[132].2   // Reserved
           TBEN_L4_8IOL:I.Data[132].3   // DXP channel 3 - Output overcurrent (ENUM bit0): 0=-, 1=active
           TBEN_L4_8IOL:I.Data[132].4   // Reserved
           TBEN_L4_8IOL:I.Data[132].5   // DXP channel 5 - Output overcurrent (ENUM bit0): 0=-, 1=active
           TBEN_L4_8IOL:I.Data[132].6   // Reserved
           TBEN_L4_8IOL:I.Data[132].7   // DXP channel 7 - Output overcurrent (ENUM bit0): 0=-, 1=active
           TBEN_L4_8IOL:I.Data[132].8   // Reserved
           TBEN_L4_8IOL:I.Data[132].9   // Reserved
           TBEN_L4_8IOL:I.Data[133]   // Port parameterization error, Wrong or missing device, Data storage error, Hardware error, Process input data invalid, Maintenance events, Out of spec. error, Parameterization error, Overtemperature, Lower limit value underrun, Upper limit value exceeded, Undervoltage, Overvoltage, Overload, Common error
           TBEN_L4_8IOL:I.Data[133].0   // Reserved
           TBEN_L4_8IOL:I.Data[133].1   // IO-Link channel 0 - Port parameterization error (ENUM bit0): 0=-, 1=active
           TBEN_L4_8IOL:I.Data[133].10   // IO-Link channel 0 - Lower limit value underrun (ENUM bit0): 0=-, 1=active
           TBEN_L4_8IOL:I.Data[133].11   // IO-Link channel 0 - Upper limit value exceeded (ENUM bit0): 0=-, 1=active
           TBEN_L4_8IOL:I.Data[133].12   // IO-Link channel 0 - Undervoltage (ENUM bit0): 0=-, 1=active
           TBEN_L4_8IOL:I.Data[133].13   // IO-Link channel 0 - Overvoltage (ENUM bit0): 0=-, 1=active
           TBEN_L4_8IOL:I.Data[133].14   // IO-Link channel 0 - Overload (ENUM bit0): 0=-, 1=active
           TBEN_L4_8IOL:I.Data[133].15   // IO-Link channel 0 - Common error (ENUM bit0): 0=-, 1=active
           TBEN_L4_8IOL:I.Data[133].2   // IO-Link channel 0 - Wrong or missing device (ENUM bit0): 0=-, 1=active
           TBEN_L4_8IOL:I.Data[133].3   // IO-Link channel 0 - Data storage error (ENUM bit0): 0=-, 1=active
           TBEN_L4_8IOL:I.Data[133].4   // IO-Link channel 0 - Hardware error (ENUM bit0): 0=-, 1=active
           TBEN_L4_8IOL:I.Data[133].5   // IO-Link channel 0 - Process input data invalid (ENUM bit0): 0=-, 1=active
           TBEN_L4_8IOL:I.Data[133].6   // IO-Link channel 0 - Maintenance events (ENUM bit0): 0=-, 1=active
           TBEN_L4_8IOL:I.Data[133].7   // IO-Link channel 0 - Out of spec. error (ENUM bit0): 0=-, 1=active
           TBEN_L4_8IOL:I.Data[133].8   // IO-Link channel 0 - Parameterization error (ENUM bit0): 0=-, 1=active
           TBEN_L4_8IOL:I.Data[133].9   // IO-Link channel 0 - Overtemperature (ENUM bit0): 0=-, 1=active
           TBEN_L4_8IOL:I.Data[134]   // Port parameterization error, Wrong or missing device, Data storage error, Hardware error, Process input data invalid, Maintenance events, Out of spec. error, Parameterization error, Overtemperature, Lower limit value underrun, Upper limit value exceeded, Undervoltage, Overvoltage, Overload, Common error
           TBEN_L4_8IOL:I.Data[134].0   // Reserved
           TBEN_L4_8IOL:I.Data[134].1   // IO-Link channel 2 - Port parameterization error (ENUM bit0): 0=-, 1=active
           TBEN_L4_8IOL:I.Data[134].10   // IO-Link channel 2 - Lower limit value underrun (ENUM bit0): 0=-, 1=active
           TBEN_L4_8IOL:I.Data[134].11   // IO-Link channel 2 - Upper limit value exceeded (ENUM bit0): 0=-, 1=active
           TBEN_L4_8IOL:I.Data[134].12   // IO-Link channel 2 - Undervoltage (ENUM bit0): 0=-, 1=active
           TBEN_L4_8IOL:I.Data[134].13   // IO-Link channel 2 - Overvoltage (ENUM bit0): 0=-, 1=active
           TBEN_L4_8IOL:I.Data[134].14   // IO-Link channel 2 - Overload (ENUM bit0): 0=-, 1=active
           TBEN_L4_8IOL:I.Data[134].15   // IO-Link channel 2 - Common error (ENUM bit0): 0=-, 1=active
           TBEN_L4_8IOL:I.Data[134].2   // IO-Link channel 2 - Wrong or missing device (ENUM bit0): 0=-, 1=active
           TBEN_L4_8IOL:I.Data[134].3   // IO-Link channel 2 - Data storage error (ENUM bit0): 0=-, 1=active
           TBEN_L4_8IOL:I.Data[134].4   // IO-Link channel 2 - Hardware error (ENUM bit0): 0=-, 1=active
           TBEN_L4_8IOL:I.Data[134].5   // IO-Link channel 2 - Process input data invalid (ENUM bit0): 0=-, 1=active
           TBEN_L4_8IOL:I.Data[134].6   // IO-Link channel 2 - Maintenance events (ENUM bit0): 0=-, 1=active
           TBEN_L4_8IOL:I.Data[134].7   // IO-Link channel 2 - Out of spec. error (ENUM bit0): 0=-, 1=active
           TBEN_L4_8IOL:I.Data[134].8   // IO-Link channel 2 - Parameterization error (ENUM bit0): 0=-, 1=active
           TBEN_L4_8IOL:I.Data[134].9   // IO-Link channel 2 - Overtemperature (ENUM bit0): 0=-, 1=active
           TBEN_L4_8IOL:I.Data[135]   // Port parameterization error, Wrong or missing device, Data storage error, Hardware error, Process input data invalid, Maintenance events, Out of spec. error, Parameterization error, Overtemperature, Lower limit value underrun, Upper limit value exceeded, Undervoltage, Overvoltage, Overload, Common error
           TBEN_L4_8IOL:I.Data[135].0   // Reserved
           TBEN_L4_8IOL:I.Data[135].1   // IO-Link channel 4 - Port parameterization error (ENUM bit0): 0=-, 1=active
           TBEN_L4_8IOL:I.Data[135].10   // IO-Link channel 4 - Lower limit value underrun (ENUM bit0): 0=-, 1=active
           TBEN_L4_8IOL:I.Data[135].11   // IO-Link channel 4 - Upper limit value exceeded (ENUM bit0): 0=-, 1=active
           TBEN_L4_8IOL:I.Data[135].12   // IO-Link channel 4 - Undervoltage (ENUM bit0): 0=-, 1=active
           TBEN_L4_8IOL:I.Data[135].13   // IO-Link channel 4 - Overvoltage (ENUM bit0): 0=-, 1=active
           TBEN_L4_8IOL:I.Data[135].14   // IO-Link channel 4 - Overload (ENUM bit0): 0=-, 1=active
           TBEN_L4_8IOL:I.Data[135].15   // IO-Link channel 4 - Common error (ENUM bit0): 0=-, 1=active
           TBEN_L4_8IOL:I.Data[135].2   // IO-Link channel 4 - Wrong or missing device (ENUM bit0): 0=-, 1=active
           TBEN_L4_8IOL:I.Data[135].3   // IO-Link channel 4 - Data storage error (ENUM bit0): 0=-, 1=active
           TBEN_L4_8IOL:I.Data[135].4   // IO-Link channel 4 - Hardware error (ENUM bit0): 0=-, 1=active
           TBEN_L4_8IOL:I.Data[135].5   // IO-Link channel 4 - Process input data invalid (ENUM bit0): 0=-, 1=active
           TBEN_L4_8IOL:I.Data[135].6   // IO-Link channel 4 - Maintenance events (ENUM bit0): 0=-, 1=active
           TBEN_L4_8IOL:I.Data[135].7   // IO-Link channel 4 - Out of spec. error (ENUM bit0): 0=-, 1=active
           TBEN_L4_8IOL:I.Data[135].8   // IO-Link channel 4 - Parameterization error (ENUM bit0): 0=-, 1=active
           TBEN_L4_8IOL:I.Data[135].9   // IO-Link channel 4 - Overtemperature (ENUM bit0): 0=-, 1=active
           TBEN_L4_8IOL:I.Data[136]   // Port parameterization error, Wrong or missing device, Data storage error, Hardware error, Process input data invalid, Maintenance events, Out of spec. error, Parameterization error, Overtemperature, Lower limit value underrun, Upper limit value exceeded, Undervoltage, Overvoltage, Overload, Common error
           TBEN_L4_8IOL:I.Data[136].0   // Reserved
           TBEN_L4_8IOL:I.Data[136].1   // IO-Link channel 6 - Port parameterization error (ENUM bit0): 0=-, 1=active
           TBEN_L4_8IOL:I.Data[136].10   // IO-Link channel 6 - Lower limit value underrun (ENUM bit0): 0=-, 1=active
           TBEN_L4_8IOL:I.Data[136].11   // IO-Link channel 6 - Upper limit value exceeded (ENUM bit0): 0=-, 1=active
           TBEN_L4_8IOL:I.Data[136].12   // IO-Link channel 6 - Undervoltage (ENUM bit0): 0=-, 1=active
           TBEN_L4_8IOL:I.Data[136].13   // IO-Link channel 6 - Overvoltage (ENUM bit0): 0=-, 1=active
           TBEN_L4_8IOL:I.Data[136].14   // IO-Link channel 6 - Overload (ENUM bit0): 0=-, 1=active
           TBEN_L4_8IOL:I.Data[136].15   // IO-Link channel 6 - Common error (ENUM bit0): 0=-, 1=active
           TBEN_L4_8IOL:I.Data[136].2   // IO-Link channel 6 - Wrong or missing device (ENUM bit0): 0=-, 1=active
           TBEN_L4_8IOL:I.Data[136].3   // IO-Link channel 6 - Data storage error (ENUM bit0): 0=-, 1=active
           TBEN_L4_8IOL:I.Data[136].4   // IO-Link channel 6 - Hardware error (ENUM bit0): 0=-, 1=active
           TBEN_L4_8IOL:I.Data[136].5   // IO-Link channel 6 - Process input data invalid (ENUM bit0): 0=-, 1=active
           TBEN_L4_8IOL:I.Data[136].6   // IO-Link channel 6 - Maintenance events (ENUM bit0): 0=-, 1=active
           TBEN_L4_8IOL:I.Data[136].7   // IO-Link channel 6 - Out of spec. error (ENUM bit0): 0=-, 1=active
           TBEN_L4_8IOL:I.Data[136].8   // IO-Link channel 6 - Parameterization error (ENUM bit0): 0=-, 1=active
           TBEN_L4_8IOL:I.Data[136].9   // IO-Link channel 6 - Overtemperature (ENUM bit0): 0=-, 1=active
           TBEN_L4_8IOL:I.Data[137]   // Port parameterization error, Wrong or missing device, Data storage error, Hardware error, Process input data invalid, Maintenance events, Out of spec. error, Parameterization error, Overtemperature, Lower limit value underrun, Upper limit value exceeded, Undervoltage, Overvoltage, Overload, Common error
           TBEN_L4_8IOL:I.Data[137].0   // Reserved
           TBEN_L4_8IOL:I.Data[137].1   // IO-Link channel 8 - Port parameterization error (ENUM bit0): 0=-, 1=active
           TBEN_L4_8IOL:I.Data[137].10   // IO-Link channel 8 - Lower limit value underrun (ENUM bit0): 0=-, 1=active
           TBEN_L4_8IOL:I.Data[137].11   // IO-Link channel 8 - Upper limit value exceeded (ENUM bit0): 0=-, 1=active
           TBEN_L4_8IOL:I.Data[137].12   // IO-Link channel 8 - Undervoltage (ENUM bit0): 0=-, 1=active
           TBEN_L4_8IOL:I.Data[137].13   // IO-Link channel 8 - Overvoltage (ENUM bit0): 0=-, 1=active
           TBEN_L4_8IOL:I.Data[137].14   // IO-Link channel 8 - Overload (ENUM bit0): 0=-, 1=active
           TBEN_L4_8IOL:I.Data[137].15   // IO-Link channel 8 - Common error (ENUM bit0): 0=-, 1=active
           TBEN_L4_8IOL:I.Data[137].2   // IO-Link channel 8 - Wrong or missing device (ENUM bit0): 0=-, 1=active
           TBEN_L4_8IOL:I.Data[137].3   // IO-Link channel 8 - Data storage error (ENUM bit0): 0=-, 1=active
           TBEN_L4_8IOL:I.Data[137].4   // IO-Link channel 8 - Hardware error (ENUM bit0): 0=-, 1=active
           TBEN_L4_8IOL:I.Data[137].5   // IO-Link channel 8 - Process input data invalid (ENUM bit0): 0=-, 1=active
           TBEN_L4_8IOL:I.Data[137].6   // IO-Link channel 8 - Maintenance events (ENUM bit0): 0=-, 1=active
           TBEN_L4_8IOL:I.Data[137].7   // IO-Link channel 8 - Out of spec. error (ENUM bit0): 0=-, 1=active
           TBEN_L4_8IOL:I.Data[137].8   // IO-Link channel 8 - Parameterization error (ENUM bit0): 0=-, 1=active
           TBEN_L4_8IOL:I.Data[137].9   // IO-Link channel 8 - Overtemperature (ENUM bit0): 0=-, 1=active
           TBEN_L4_8IOL:I.Data[138]   // Port parameterization error, Wrong or missing device, Data storage error, Hardware error, Process input data invalid, Maintenance events, Out of spec. error, Parameterization error, Overtemperature, Lower limit value underrun, Upper limit value exceeded, Undervoltage, Overvoltage, Overload, Common error
           TBEN_L4_8IOL:I.Data[138].0   // Reserved
           TBEN_L4_8IOL:I.Data[138].1   // IO-Link channel 10 - Port parameterization error (ENUM bit0): 0=-, 1=active
           TBEN_L4_8IOL:I.Data[138].10   // IO-Link channel 10 - Lower limit value underrun (ENUM bit0): 0=-, 1=active
           TBEN_L4_8IOL:I.Data[138].11   // IO-Link channel 10 - Upper limit value exceeded (ENUM bit0): 0=-, 1=active
           TBEN_L4_8IOL:I.Data[138].12   // IO-Link channel 10 - Undervoltage (ENUM bit0): 0=-, 1=active
           TBEN_L4_8IOL:I.Data[138].13   // IO-Link channel 10 - Overvoltage (ENUM bit0): 0=-, 1=active
           TBEN_L4_8IOL:I.Data[138].14   // IO-Link channel 10 - Overload (ENUM bit0): 0=-, 1=active
           TBEN_L4_8IOL:I.Data[138].15   // IO-Link channel 10 - Common error (ENUM bit0): 0=-, 1=active
           TBEN_L4_8IOL:I.Data[138].2   // IO-Link channel 10 - Wrong or missing device (ENUM bit0): 0=-, 1=active
           TBEN_L4_8IOL:I.Data[138].3   // IO-Link channel 10 - Data storage error (ENUM bit0): 0=-, 1=active
           TBEN_L4_8IOL:I.Data[138].4   // IO-Link channel 10 - Hardware error (ENUM bit0): 0=-, 1=active
           TBEN_L4_8IOL:I.Data[138].5   // IO-Link channel 10 - Process input data invalid (ENUM bit0): 0=-, 1=active
           TBEN_L4_8IOL:I.Data[138].6   // IO-Link channel 10 - Maintenance events (ENUM bit0): 0=-, 1=active
           TBEN_L4_8IOL:I.Data[138].7   // IO-Link channel 10 - Out of spec. error (ENUM bit0): 0=-, 1=active
           TBEN_L4_8IOL:I.Data[138].8   // IO-Link channel 10 - Parameterization error (ENUM bit0): 0=-, 1=active
           TBEN_L4_8IOL:I.Data[138].9   // IO-Link channel 10 - Overtemperature (ENUM bit0): 0=-, 1=active
           TBEN_L4_8IOL:I.Data[139]   // Port parameterization error, Wrong or missing device, Data storage error, Hardware error, Process input data invalid, Maintenance events, Out of spec. error, Parameterization error, Overtemperature, Lower limit value underrun, Upper limit value exceeded, Undervoltage, Overvoltage, Overload, Common error
           TBEN_L4_8IOL:I.Data[139].0   // Reserved
           TBEN_L4_8IOL:I.Data[139].1   // IO-Link channel 12 - Port parameterization error (ENUM bit0): 0=-, 1=active
           TBEN_L4_8IOL:I.Data[139].10   // IO-Link channel 12 - Lower limit value underrun (ENUM bit0): 0=-, 1=active
           TBEN_L4_8IOL:I.Data[139].11   // IO-Link channel 12 - Upper limit value exceeded (ENUM bit0): 0=-, 1=active
           TBEN_L4_8IOL:I.Data[139].12   // IO-Link channel 12 - Undervoltage (ENUM bit0): 0=-, 1=active
           TBEN_L4_8IOL:I.Data[139].13   // IO-Link channel 12 - Overvoltage (ENUM bit0): 0=-, 1=active
           TBEN_L4_8IOL:I.Data[139].14   // IO-Link channel 12 - Overload (ENUM bit0): 0=-, 1=active
           TBEN_L4_8IOL:I.Data[139].15   // IO-Link channel 12 - Common error (ENUM bit0): 0=-, 1=active
           TBEN_L4_8IOL:I.Data[139].2   // IO-Link channel 12 - Wrong or missing device (ENUM bit0): 0=-, 1=active
           TBEN_L4_8IOL:I.Data[139].3   // IO-Link channel 12 - Data storage error (ENUM bit0): 0=-, 1=active
           TBEN_L4_8IOL:I.Data[139].4   // IO-Link channel 12 - Hardware error (ENUM bit0): 0=-, 1=active
           TBEN_L4_8IOL:I.Data[139].5   // IO-Link channel 12 - Process input data invalid (ENUM bit0): 0=-, 1=active
           TBEN_L4_8IOL:I.Data[139].6   // IO-Link channel 12 - Maintenance events (ENUM bit0): 0=-, 1=active
           TBEN_L4_8IOL:I.Data[139].7   // IO-Link channel 12 - Out of spec. error (ENUM bit0): 0=-, 1=active
           TBEN_L4_8IOL:I.Data[139].8   // IO-Link channel 12 - Parameterization error (ENUM bit0): 0=-, 1=active
           TBEN_L4_8IOL:I.Data[139].9   // IO-Link channel 12 - Overtemperature (ENUM bit0): 0=-, 1=active
           TBEN_L4_8IOL:I.Data[13]   // IO-Link Port 1 - Input data word 10
           TBEN_L4_8IOL:I.Data[13].0   // IO-Link Port 1 - Input data word 10 (INT bit0)
           TBEN_L4_8IOL:I.Data[13].1   // IO-Link Port 1 - Input data word 10 (INT bit1)
           TBEN_L4_8IOL:I.Data[13].10   // IO-Link Port 1 - Input data word 10 (INT bit10)
           TBEN_L4_8IOL:I.Data[13].11   // IO-Link Port 1 - Input data word 10 (INT bit11)
           TBEN_L4_8IOL:I.Data[13].12   // IO-Link Port 1 - Input data word 10 (INT bit12)
           TBEN_L4_8IOL:I.Data[13].13   // IO-Link Port 1 - Input data word 10 (INT bit13)
           TBEN_L4_8IOL:I.Data[13].14   // IO-Link Port 1 - Input data word 10 (INT bit14)
           TBEN_L4_8IOL:I.Data[13].15   // IO-Link Port 1 - Input data word 10 (INT bit15)
           TBEN_L4_8IOL:I.Data[13].2   // IO-Link Port 1 - Input data word 10 (INT bit2)
           TBEN_L4_8IOL:I.Data[13].3   // IO-Link Port 1 - Input data word 10 (INT bit3)
           TBEN_L4_8IOL:I.Data[13].4   // IO-Link Port 1 - Input data word 10 (INT bit4)
           TBEN_L4_8IOL:I.Data[13].5   // IO-Link Port 1 - Input data word 10 (INT bit5)
           TBEN_L4_8IOL:I.Data[13].6   // IO-Link Port 1 - Input data word 10 (INT bit6)
           TBEN_L4_8IOL:I.Data[13].7   // IO-Link Port 1 - Input data word 10 (INT bit7)
           TBEN_L4_8IOL:I.Data[13].8   // IO-Link Port 1 - Input data word 10 (INT bit8)
           TBEN_L4_8IOL:I.Data[13].9   // IO-Link Port 1 - Input data word 10 (INT bit9)
           TBEN_L4_8IOL:I.Data[140]   // Port parameterization error, Wrong or missing device, Data storage error, Hardware error, Process input data invalid, Maintenance events, Out of spec. error, Parameterization error, Overtemperature, Lower limit value underrun, Upper limit value exceeded, Undervoltage, Overvoltage, Overload, Common error
           TBEN_L4_8IOL:I.Data[140].0   // Reserved
           TBEN_L4_8IOL:I.Data[140].1   // IO-Link channel 14 - Port parameterization error (ENUM bit0): 0=-, 1=active
           TBEN_L4_8IOL:I.Data[140].10   // IO-Link channel 14 - Lower limit value underrun (ENUM bit0): 0=-, 1=active
           TBEN_L4_8IOL:I.Data[140].11   // IO-Link channel 14 - Upper limit value exceeded (ENUM bit0): 0=-, 1=active
           TBEN_L4_8IOL:I.Data[140].12   // IO-Link channel 14 - Undervoltage (ENUM bit0): 0=-, 1=active
           TBEN_L4_8IOL:I.Data[140].13   // IO-Link channel 14 - Overvoltage (ENUM bit0): 0=-, 1=active
           TBEN_L4_8IOL:I.Data[140].14   // IO-Link channel 14 - Overload (ENUM bit0): 0=-, 1=active
           TBEN_L4_8IOL:I.Data[140].15   // IO-Link channel 14 - Common error (ENUM bit0): 0=-, 1=active
           TBEN_L4_8IOL:I.Data[140].2   // IO-Link channel 14 - Wrong or missing device (ENUM bit0): 0=-, 1=active
           TBEN_L4_8IOL:I.Data[140].3   // IO-Link channel 14 - Data storage error (ENUM bit0): 0=-, 1=active
           TBEN_L4_8IOL:I.Data[140].4   // IO-Link channel 14 - Hardware error (ENUM bit0): 0=-, 1=active
           TBEN_L4_8IOL:I.Data[140].5   // IO-Link channel 14 - Process input data invalid (ENUM bit0): 0=-, 1=active
           TBEN_L4_8IOL:I.Data[140].6   // IO-Link channel 14 - Maintenance events (ENUM bit0): 0=-, 1=active
           TBEN_L4_8IOL:I.Data[140].7   // IO-Link channel 14 - Out of spec. error (ENUM bit0): 0=-, 1=active
           TBEN_L4_8IOL:I.Data[140].8   // IO-Link channel 14 - Parameterization error (ENUM bit0): 0=-, 1=active
           TBEN_L4_8IOL:I.Data[140].9   // IO-Link channel 14 - Overtemperature (ENUM bit0): 0=-, 1=active
           TBEN_L4_8IOL:I.Data[141]   // IO-Link event 1 - Qualifier, IO-Link event 1 - Port
           TBEN_L4_8IOL:I.Data[141].0   // IO-Link event 1 - Qualifier (INT bit0)
           TBEN_L4_8IOL:I.Data[141].1   // IO-Link event 1 - Qualifier (INT bit1)
           TBEN_L4_8IOL:I.Data[141].10   // IO-Link event 1 - Port (INT bit2)
           TBEN_L4_8IOL:I.Data[141].11   // IO-Link event 1 - Port (INT bit3)
           TBEN_L4_8IOL:I.Data[141].12   // IO-Link event 1 - Port (INT bit4)
           TBEN_L4_8IOL:I.Data[141].13   // IO-Link event 1 - Port (INT bit5)
           TBEN_L4_8IOL:I.Data[141].14   // IO-Link event 1 - Port (INT bit6)
           TBEN_L4_8IOL:I.Data[141].15   // IO-Link event 1 - Port (INT bit7)
           TBEN_L4_8IOL:I.Data[141].2   // IO-Link event 1 - Qualifier (INT bit2)
           TBEN_L4_8IOL:I.Data[141].3   // IO-Link event 1 - Qualifier (INT bit3)
           TBEN_L4_8IOL:I.Data[141].4   // IO-Link event 1 - Qualifier (INT bit4)
           TBEN_L4_8IOL:I.Data[141].5   // IO-Link event 1 - Qualifier (INT bit5)
           TBEN_L4_8IOL:I.Data[141].6   // IO-Link event 1 - Qualifier (INT bit6)
           TBEN_L4_8IOL:I.Data[141].7   // IO-Link event 1 - Qualifier (INT bit7)
           TBEN_L4_8IOL:I.Data[141].8   // IO-Link event 1 - Port (INT bit0)
           TBEN_L4_8IOL:I.Data[141].9   // IO-Link event 1 - Port (INT bit1)
           TBEN_L4_8IOL:I.Data[142]   // IO-Link event 1 - Event code
           TBEN_L4_8IOL:I.Data[142].0   // IO-Link event 1 - Event code (INT bit0)
           TBEN_L4_8IOL:I.Data[142].1   // IO-Link event 1 - Event code (INT bit1)
           TBEN_L4_8IOL:I.Data[142].10   // IO-Link event 1 - Event code (INT bit10)
           TBEN_L4_8IOL:I.Data[142].11   // IO-Link event 1 - Event code (INT bit11)
           TBEN_L4_8IOL:I.Data[142].12   // IO-Link event 1 - Event code (INT bit12)
           TBEN_L4_8IOL:I.Data[142].13   // IO-Link event 1 - Event code (INT bit13)
           TBEN_L4_8IOL:I.Data[142].14   // IO-Link event 1 - Event code (INT bit14)
           TBEN_L4_8IOL:I.Data[142].15   // IO-Link event 1 - Event code (INT bit15)
           TBEN_L4_8IOL:I.Data[142].2   // IO-Link event 1 - Event code (INT bit2)
           TBEN_L4_8IOL:I.Data[142].3   // IO-Link event 1 - Event code (INT bit3)
           TBEN_L4_8IOL:I.Data[142].4   // IO-Link event 1 - Event code (INT bit4)
           TBEN_L4_8IOL:I.Data[142].5   // IO-Link event 1 - Event code (INT bit5)
           TBEN_L4_8IOL:I.Data[142].6   // IO-Link event 1 - Event code (INT bit6)
           TBEN_L4_8IOL:I.Data[142].7   // IO-Link event 1 - Event code (INT bit7)
           TBEN_L4_8IOL:I.Data[142].8   // IO-Link event 1 - Event code (INT bit8)
           TBEN_L4_8IOL:I.Data[142].9   // IO-Link event 1 - Event code (INT bit9)
           TBEN_L4_8IOL:I.Data[143]   // IO-Link event 2 - Qualifier, IO-Link event 2 - Port
           TBEN_L4_8IOL:I.Data[143].0   // IO-Link event 2 - Qualifier (INT bit0)
           TBEN_L4_8IOL:I.Data[143].1   // IO-Link event 2 - Qualifier (INT bit1)
           TBEN_L4_8IOL:I.Data[143].10   // IO-Link event 2 - Port (INT bit2)
           TBEN_L4_8IOL:I.Data[143].11   // IO-Link event 2 - Port (INT bit3)
           TBEN_L4_8IOL:I.Data[143].12   // IO-Link event 2 - Port (INT bit4)
           TBEN_L4_8IOL:I.Data[143].13   // IO-Link event 2 - Port (INT bit5)
           TBEN_L4_8IOL:I.Data[143].14   // IO-Link event 2 - Port (INT bit6)
           TBEN_L4_8IOL:I.Data[143].15   // IO-Link event 2 - Port (INT bit7)
           TBEN_L4_8IOL:I.Data[143].2   // IO-Link event 2 - Qualifier (INT bit2)
           TBEN_L4_8IOL:I.Data[143].3   // IO-Link event 2 - Qualifier (INT bit3)
           TBEN_L4_8IOL:I.Data[143].4   // IO-Link event 2 - Qualifier (INT bit4)
           TBEN_L4_8IOL:I.Data[143].5   // IO-Link event 2 - Qualifier (INT bit5)
           TBEN_L4_8IOL:I.Data[143].6   // IO-Link event 2 - Qualifier (INT bit6)
           TBEN_L4_8IOL:I.Data[143].7   // IO-Link event 2 - Qualifier (INT bit7)
           TBEN_L4_8IOL:I.Data[143].8   // IO-Link event 2 - Port (INT bit0)
           TBEN_L4_8IOL:I.Data[143].9   // IO-Link event 2 - Port (INT bit1)
           TBEN_L4_8IOL:I.Data[144]   // IO-Link event 2 - Event code
           TBEN_L4_8IOL:I.Data[144].0   // IO-Link event 2 - Event code (INT bit0)
           TBEN_L4_8IOL:I.Data[144].1   // IO-Link event 2 - Event code (INT bit1)
           TBEN_L4_8IOL:I.Data[144].10   // IO-Link event 2 - Event code (INT bit10)
           TBEN_L4_8IOL:I.Data[144].11   // IO-Link event 2 - Event code (INT bit11)
           TBEN_L4_8IOL:I.Data[144].12   // IO-Link event 2 - Event code (INT bit12)
           TBEN_L4_8IOL:I.Data[144].13   // IO-Link event 2 - Event code (INT bit13)
           TBEN_L4_8IOL:I.Data[144].14   // IO-Link event 2 - Event code (INT bit14)
           TBEN_L4_8IOL:I.Data[144].15   // IO-Link event 2 - Event code (INT bit15)
           TBEN_L4_8IOL:I.Data[144].2   // IO-Link event 2 - Event code (INT bit2)
           TBEN_L4_8IOL:I.Data[144].3   // IO-Link event 2 - Event code (INT bit3)
           TBEN_L4_8IOL:I.Data[144].4   // IO-Link event 2 - Event code (INT bit4)
           TBEN_L4_8IOL:I.Data[144].5   // IO-Link event 2 - Event code (INT bit5)
           TBEN_L4_8IOL:I.Data[144].6   // IO-Link event 2 - Event code (INT bit6)
           TBEN_L4_8IOL:I.Data[144].7   // IO-Link event 2 - Event code (INT bit7)
           TBEN_L4_8IOL:I.Data[144].8   // IO-Link event 2 - Event code (INT bit8)
           TBEN_L4_8IOL:I.Data[144].9   // IO-Link event 2 - Event code (INT bit9)
           TBEN_L4_8IOL:I.Data[145]   // IO-Link event 3 - Qualifier, IO-Link event 3 - Port
           TBEN_L4_8IOL:I.Data[145].0   // IO-Link event 3 - Qualifier (INT bit0)
           TBEN_L4_8IOL:I.Data[145].1   // IO-Link event 3 - Qualifier (INT bit1)
           TBEN_L4_8IOL:I.Data[145].10   // IO-Link event 3 - Port (INT bit2)
           TBEN_L4_8IOL:I.Data[145].11   // IO-Link event 3 - Port (INT bit3)
           TBEN_L4_8IOL:I.Data[145].12   // IO-Link event 3 - Port (INT bit4)
           TBEN_L4_8IOL:I.Data[145].13   // IO-Link event 3 - Port (INT bit5)
           TBEN_L4_8IOL:I.Data[145].14   // IO-Link event 3 - Port (INT bit6)
           TBEN_L4_8IOL:I.Data[145].15   // IO-Link event 3 - Port (INT bit7)
           TBEN_L4_8IOL:I.Data[145].2   // IO-Link event 3 - Qualifier (INT bit2)
           TBEN_L4_8IOL:I.Data[145].3   // IO-Link event 3 - Qualifier (INT bit3)
           TBEN_L4_8IOL:I.Data[145].4   // IO-Link event 3 - Qualifier (INT bit4)
           TBEN_L4_8IOL:I.Data[145].5   // IO-Link event 3 - Qualifier (INT bit5)
           TBEN_L4_8IOL:I.Data[145].6   // IO-Link event 3 - Qualifier (INT bit6)
           TBEN_L4_8IOL:I.Data[145].7   // IO-Link event 3 - Qualifier (INT bit7)
           TBEN_L4_8IOL:I.Data[145].8   // IO-Link event 3 - Port (INT bit0)
           TBEN_L4_8IOL:I.Data[145].9   // IO-Link event 3 - Port (INT bit1)
           TBEN_L4_8IOL:I.Data[146]   // IO-Link event 3 - Event code
           TBEN_L4_8IOL:I.Data[146].0   // IO-Link event 3 - Event code (INT bit0)
           TBEN_L4_8IOL:I.Data[146].1   // IO-Link event 3 - Event code (INT bit1)
           TBEN_L4_8IOL:I.Data[146].10   // IO-Link event 3 - Event code (INT bit10)
           TBEN_L4_8IOL:I.Data[146].11   // IO-Link event 3 - Event code (INT bit11)
           TBEN_L4_8IOL:I.Data[146].12   // IO-Link event 3 - Event code (INT bit12)
           TBEN_L4_8IOL:I.Data[146].13   // IO-Link event 3 - Event code (INT bit13)
           TBEN_L4_8IOL:I.Data[146].14   // IO-Link event 3 - Event code (INT bit14)
           TBEN_L4_8IOL:I.Data[146].15   // IO-Link event 3 - Event code (INT bit15)
           TBEN_L4_8IOL:I.Data[146].2   // IO-Link event 3 - Event code (INT bit2)
           TBEN_L4_8IOL:I.Data[146].3   // IO-Link event 3 - Event code (INT bit3)
           TBEN_L4_8IOL:I.Data[146].4   // IO-Link event 3 - Event code (INT bit4)
           TBEN_L4_8IOL:I.Data[146].5   // IO-Link event 3 - Event code (INT bit5)
           TBEN_L4_8IOL:I.Data[146].6   // IO-Link event 3 - Event code (INT bit6)
           TBEN_L4_8IOL:I.Data[146].7   // IO-Link event 3 - Event code (INT bit7)
           TBEN_L4_8IOL:I.Data[146].8   // IO-Link event 3 - Event code (INT bit8)
           TBEN_L4_8IOL:I.Data[146].9   // IO-Link event 3 - Event code (INT bit9)
           TBEN_L4_8IOL:I.Data[147]   // IO-Link event 4 - Qualifier, IO-Link event 4 - Port
           TBEN_L4_8IOL:I.Data[147].0   // IO-Link event 4 - Qualifier (INT bit0)
           TBEN_L4_8IOL:I.Data[147].1   // IO-Link event 4 - Qualifier (INT bit1)
           TBEN_L4_8IOL:I.Data[147].10   // IO-Link event 4 - Port (INT bit2)
           TBEN_L4_8IOL:I.Data[147].11   // IO-Link event 4 - Port (INT bit3)
           TBEN_L4_8IOL:I.Data[147].12   // IO-Link event 4 - Port (INT bit4)
           TBEN_L4_8IOL:I.Data[147].13   // IO-Link event 4 - Port (INT bit5)
           TBEN_L4_8IOL:I.Data[147].14   // IO-Link event 4 - Port (INT bit6)
           TBEN_L4_8IOL:I.Data[147].15   // IO-Link event 4 - Port (INT bit7)
           TBEN_L4_8IOL:I.Data[147].2   // IO-Link event 4 - Qualifier (INT bit2)
           TBEN_L4_8IOL:I.Data[147].3   // IO-Link event 4 - Qualifier (INT bit3)
           TBEN_L4_8IOL:I.Data[147].4   // IO-Link event 4 - Qualifier (INT bit4)
           TBEN_L4_8IOL:I.Data[147].5   // IO-Link event 4 - Qualifier (INT bit5)
           TBEN_L4_8IOL:I.Data[147].6   // IO-Link event 4 - Qualifier (INT bit6)
           TBEN_L4_8IOL:I.Data[147].7   // IO-Link event 4 - Qualifier (INT bit7)
           TBEN_L4_8IOL:I.Data[147].8   // IO-Link event 4 - Port (INT bit0)
           TBEN_L4_8IOL:I.Data[147].9   // IO-Link event 4 - Port (INT bit1)
           TBEN_L4_8IOL:I.Data[148]   // IO-Link event 4 - Event code
           TBEN_L4_8IOL:I.Data[148].0   // IO-Link event 4 - Event code (INT bit0)
           TBEN_L4_8IOL:I.Data[148].1   // IO-Link event 4 - Event code (INT bit1)
           TBEN_L4_8IOL:I.Data[148].10   // IO-Link event 4 - Event code (INT bit10)
           TBEN_L4_8IOL:I.Data[148].11   // IO-Link event 4 - Event code (INT bit11)
           TBEN_L4_8IOL:I.Data[148].12   // IO-Link event 4 - Event code (INT bit12)
           TBEN_L4_8IOL:I.Data[148].13   // IO-Link event 4 - Event code (INT bit13)
           TBEN_L4_8IOL:I.Data[148].14   // IO-Link event 4 - Event code (INT bit14)
           TBEN_L4_8IOL:I.Data[148].15   // IO-Link event 4 - Event code (INT bit15)
           TBEN_L4_8IOL:I.Data[148].2   // IO-Link event 4 - Event code (INT bit2)
           TBEN_L4_8IOL:I.Data[148].3   // IO-Link event 4 - Event code (INT bit3)
           TBEN_L4_8IOL:I.Data[148].4   // IO-Link event 4 - Event code (INT bit4)
           TBEN_L4_8IOL:I.Data[148].5   // IO-Link event 4 - Event code (INT bit5)
           TBEN_L4_8IOL:I.Data[148].6   // IO-Link event 4 - Event code (INT bit6)
           TBEN_L4_8IOL:I.Data[148].7   // IO-Link event 4 - Event code (INT bit7)
           TBEN_L4_8IOL:I.Data[148].8   // IO-Link event 4 - Event code (INT bit8)
           TBEN_L4_8IOL:I.Data[148].9   // IO-Link event 4 - Event code (INT bit9)
           TBEN_L4_8IOL:I.Data[149]   // IO-Link event 5 - Qualifier, IO-Link event 5 - Port
           TBEN_L4_8IOL:I.Data[149].0   // IO-Link event 5 - Qualifier (INT bit0)
           TBEN_L4_8IOL:I.Data[149].1   // IO-Link event 5 - Qualifier (INT bit1)
           TBEN_L4_8IOL:I.Data[149].10   // IO-Link event 5 - Port (INT bit2)
           TBEN_L4_8IOL:I.Data[149].11   // IO-Link event 5 - Port (INT bit3)
           TBEN_L4_8IOL:I.Data[149].12   // IO-Link event 5 - Port (INT bit4)
           TBEN_L4_8IOL:I.Data[149].13   // IO-Link event 5 - Port (INT bit5)
           TBEN_L4_8IOL:I.Data[149].14   // IO-Link event 5 - Port (INT bit6)
           TBEN_L4_8IOL:I.Data[149].15   // IO-Link event 5 - Port (INT bit7)
           TBEN_L4_8IOL:I.Data[149].2   // IO-Link event 5 - Qualifier (INT bit2)
           TBEN_L4_8IOL:I.Data[149].3   // IO-Link event 5 - Qualifier (INT bit3)
           TBEN_L4_8IOL:I.Data[149].4   // IO-Link event 5 - Qualifier (INT bit4)
           TBEN_L4_8IOL:I.Data[149].5   // IO-Link event 5 - Qualifier (INT bit5)
           TBEN_L4_8IOL:I.Data[149].6   // IO-Link event 5 - Qualifier (INT bit6)
           TBEN_L4_8IOL:I.Data[149].7   // IO-Link event 5 - Qualifier (INT bit7)
           TBEN_L4_8IOL:I.Data[149].8   // IO-Link event 5 - Port (INT bit0)
           TBEN_L4_8IOL:I.Data[149].9   // IO-Link event 5 - Port (INT bit1)
           TBEN_L4_8IOL:I.Data[14]   // IO-Link Port 1 - Input data word 11
           TBEN_L4_8IOL:I.Data[14].0   // IO-Link Port 1 - Input data word 11 (INT bit0)
           TBEN_L4_8IOL:I.Data[14].1   // IO-Link Port 1 - Input data word 11 (INT bit1)
           TBEN_L4_8IOL:I.Data[14].10   // IO-Link Port 1 - Input data word 11 (INT bit10)
           TBEN_L4_8IOL:I.Data[14].11   // IO-Link Port 1 - Input data word 11 (INT bit11)
           TBEN_L4_8IOL:I.Data[14].12   // IO-Link Port 1 - Input data word 11 (INT bit12)
           TBEN_L4_8IOL:I.Data[14].13   // IO-Link Port 1 - Input data word 11 (INT bit13)
           TBEN_L4_8IOL:I.Data[14].14   // IO-Link Port 1 - Input data word 11 (INT bit14)
           TBEN_L4_8IOL:I.Data[14].15   // IO-Link Port 1 - Input data word 11 (INT bit15)
           TBEN_L4_8IOL:I.Data[14].2   // IO-Link Port 1 - Input data word 11 (INT bit2)
           TBEN_L4_8IOL:I.Data[14].3   // IO-Link Port 1 - Input data word 11 (INT bit3)
           TBEN_L4_8IOL:I.Data[14].4   // IO-Link Port 1 - Input data word 11 (INT bit4)
           TBEN_L4_8IOL:I.Data[14].5   // IO-Link Port 1 - Input data word 11 (INT bit5)
           TBEN_L4_8IOL:I.Data[14].6   // IO-Link Port 1 - Input data word 11 (INT bit6)
           TBEN_L4_8IOL:I.Data[14].7   // IO-Link Port 1 - Input data word 11 (INT bit7)
           TBEN_L4_8IOL:I.Data[14].8   // IO-Link Port 1 - Input data word 11 (INT bit8)
           TBEN_L4_8IOL:I.Data[14].9   // IO-Link Port 1 - Input data word 11 (INT bit9)
           TBEN_L4_8IOL:I.Data[150]   // IO-Link event 5 - Event code
           TBEN_L4_8IOL:I.Data[150].0   // IO-Link event 5 - Event code (INT bit0)
           TBEN_L4_8IOL:I.Data[150].1   // IO-Link event 5 - Event code (INT bit1)
           TBEN_L4_8IOL:I.Data[150].10   // IO-Link event 5 - Event code (INT bit10)
           TBEN_L4_8IOL:I.Data[150].11   // IO-Link event 5 - Event code (INT bit11)
           TBEN_L4_8IOL:I.Data[150].12   // IO-Link event 5 - Event code (INT bit12)
           TBEN_L4_8IOL:I.Data[150].13   // IO-Link event 5 - Event code (INT bit13)
           TBEN_L4_8IOL:I.Data[150].14   // IO-Link event 5 - Event code (INT bit14)
           TBEN_L4_8IOL:I.Data[150].15   // IO-Link event 5 - Event code (INT bit15)
           TBEN_L4_8IOL:I.Data[150].2   // IO-Link event 5 - Event code (INT bit2)
           TBEN_L4_8IOL:I.Data[150].3   // IO-Link event 5 - Event code (INT bit3)
           TBEN_L4_8IOL:I.Data[150].4   // IO-Link event 5 - Event code (INT bit4)
           TBEN_L4_8IOL:I.Data[150].5   // IO-Link event 5 - Event code (INT bit5)
           TBEN_L4_8IOL:I.Data[150].6   // IO-Link event 5 - Event code (INT bit6)
           TBEN_L4_8IOL:I.Data[150].7   // IO-Link event 5 - Event code (INT bit7)
           TBEN_L4_8IOL:I.Data[150].8   // IO-Link event 5 - Event code (INT bit8)
           TBEN_L4_8IOL:I.Data[150].9   // IO-Link event 5 - Event code (INT bit9)
           TBEN_L4_8IOL:I.Data[151]   // IO-Link event 6 - Qualifier, IO-Link event 6 - Port
           TBEN_L4_8IOL:I.Data[151].0   // IO-Link event 6 - Qualifier (INT bit0)
           TBEN_L4_8IOL:I.Data[151].1   // IO-Link event 6 - Qualifier (INT bit1)
           TBEN_L4_8IOL:I.Data[151].10   // IO-Link event 6 - Port (INT bit2)
           TBEN_L4_8IOL:I.Data[151].11   // IO-Link event 6 - Port (INT bit3)
           TBEN_L4_8IOL:I.Data[151].12   // IO-Link event 6 - Port (INT bit4)
           TBEN_L4_8IOL:I.Data[151].13   // IO-Link event 6 - Port (INT bit5)
           TBEN_L4_8IOL:I.Data[151].14   // IO-Link event 6 - Port (INT bit6)
           TBEN_L4_8IOL:I.Data[151].15   // IO-Link event 6 - Port (INT bit7)
           TBEN_L4_8IOL:I.Data[151].2   // IO-Link event 6 - Qualifier (INT bit2)
           TBEN_L4_8IOL:I.Data[151].3   // IO-Link event 6 - Qualifier (INT bit3)
           TBEN_L4_8IOL:I.Data[151].4   // IO-Link event 6 - Qualifier (INT bit4)
           TBEN_L4_8IOL:I.Data[151].5   // IO-Link event 6 - Qualifier (INT bit5)
           TBEN_L4_8IOL:I.Data[151].6   // IO-Link event 6 - Qualifier (INT bit6)
           TBEN_L4_8IOL:I.Data[151].7   // IO-Link event 6 - Qualifier (INT bit7)
           TBEN_L4_8IOL:I.Data[151].8   // IO-Link event 6 - Port (INT bit0)
           TBEN_L4_8IOL:I.Data[151].9   // IO-Link event 6 - Port (INT bit1)
           TBEN_L4_8IOL:I.Data[152]   // IO-Link event 6 - Event code
           TBEN_L4_8IOL:I.Data[152].0   // IO-Link event 6 - Event code (INT bit0)
           TBEN_L4_8IOL:I.Data[152].1   // IO-Link event 6 - Event code (INT bit1)
           TBEN_L4_8IOL:I.Data[152].10   // IO-Link event 6 - Event code (INT bit10)
           TBEN_L4_8IOL:I.Data[152].11   // IO-Link event 6 - Event code (INT bit11)
           TBEN_L4_8IOL:I.Data[152].12   // IO-Link event 6 - Event code (INT bit12)
           TBEN_L4_8IOL:I.Data[152].13   // IO-Link event 6 - Event code (INT bit13)
           TBEN_L4_8IOL:I.Data[152].14   // IO-Link event 6 - Event code (INT bit14)
           TBEN_L4_8IOL:I.Data[152].15   // IO-Link event 6 - Event code (INT bit15)
           TBEN_L4_8IOL:I.Data[152].2   // IO-Link event 6 - Event code (INT bit2)
           TBEN_L4_8IOL:I.Data[152].3   // IO-Link event 6 - Event code (INT bit3)
           TBEN_L4_8IOL:I.Data[152].4   // IO-Link event 6 - Event code (INT bit4)
           TBEN_L4_8IOL:I.Data[152].5   // IO-Link event 6 - Event code (INT bit5)
           TBEN_L4_8IOL:I.Data[152].6   // IO-Link event 6 - Event code (INT bit6)
           TBEN_L4_8IOL:I.Data[152].7   // IO-Link event 6 - Event code (INT bit7)
           TBEN_L4_8IOL:I.Data[152].8   // IO-Link event 6 - Event code (INT bit8)
           TBEN_L4_8IOL:I.Data[152].9   // IO-Link event 6 - Event code (INT bit9)
           TBEN_L4_8IOL:I.Data[153]   // IO-Link event 7 - Qualifier, IO-Link event 7 - Port
           TBEN_L4_8IOL:I.Data[153].0   // IO-Link event 7 - Qualifier (INT bit0)
           TBEN_L4_8IOL:I.Data[153].1   // IO-Link event 7 - Qualifier (INT bit1)
           TBEN_L4_8IOL:I.Data[153].10   // IO-Link event 7 - Port (INT bit2)
           TBEN_L4_8IOL:I.Data[153].11   // IO-Link event 7 - Port (INT bit3)
           TBEN_L4_8IOL:I.Data[153].12   // IO-Link event 7 - Port (INT bit4)
           TBEN_L4_8IOL:I.Data[153].13   // IO-Link event 7 - Port (INT bit5)
           TBEN_L4_8IOL:I.Data[153].14   // IO-Link event 7 - Port (INT bit6)
           TBEN_L4_8IOL:I.Data[153].15   // IO-Link event 7 - Port (INT bit7)
           TBEN_L4_8IOL:I.Data[153].2   // IO-Link event 7 - Qualifier (INT bit2)
           TBEN_L4_8IOL:I.Data[153].3   // IO-Link event 7 - Qualifier (INT bit3)
           TBEN_L4_8IOL:I.Data[153].4   // IO-Link event 7 - Qualifier (INT bit4)
           TBEN_L4_8IOL:I.Data[153].5   // IO-Link event 7 - Qualifier (INT bit5)
           TBEN_L4_8IOL:I.Data[153].6   // IO-Link event 7 - Qualifier (INT bit6)
           TBEN_L4_8IOL:I.Data[153].7   // IO-Link event 7 - Qualifier (INT bit7)
           TBEN_L4_8IOL:I.Data[153].8   // IO-Link event 7 - Port (INT bit0)
           TBEN_L4_8IOL:I.Data[153].9   // IO-Link event 7 - Port (INT bit1)
           TBEN_L4_8IOL:I.Data[154]   // IO-Link event 7 - Event code
           TBEN_L4_8IOL:I.Data[154].0   // IO-Link event 7 - Event code (INT bit0)
           TBEN_L4_8IOL:I.Data[154].1   // IO-Link event 7 - Event code (INT bit1)
           TBEN_L4_8IOL:I.Data[154].10   // IO-Link event 7 - Event code (INT bit10)
           TBEN_L4_8IOL:I.Data[154].11   // IO-Link event 7 - Event code (INT bit11)
           TBEN_L4_8IOL:I.Data[154].12   // IO-Link event 7 - Event code (INT bit12)
           TBEN_L4_8IOL:I.Data[154].13   // IO-Link event 7 - Event code (INT bit13)
           TBEN_L4_8IOL:I.Data[154].14   // IO-Link event 7 - Event code (INT bit14)
           TBEN_L4_8IOL:I.Data[154].15   // IO-Link event 7 - Event code (INT bit15)
           TBEN_L4_8IOL:I.Data[154].2   // IO-Link event 7 - Event code (INT bit2)
           TBEN_L4_8IOL:I.Data[154].3   // IO-Link event 7 - Event code (INT bit3)
           TBEN_L4_8IOL:I.Data[154].4   // IO-Link event 7 - Event code (INT bit4)
           TBEN_L4_8IOL:I.Data[154].5   // IO-Link event 7 - Event code (INT bit5)
           TBEN_L4_8IOL:I.Data[154].6   // IO-Link event 7 - Event code (INT bit6)
           TBEN_L4_8IOL:I.Data[154].7   // IO-Link event 7 - Event code (INT bit7)
           TBEN_L4_8IOL:I.Data[154].8   // IO-Link event 7 - Event code (INT bit8)
           TBEN_L4_8IOL:I.Data[154].9   // IO-Link event 7 - Event code (INT bit9)
           TBEN_L4_8IOL:I.Data[155]   // IO-Link event 8 - Qualifier, IO-Link event 8 - Port
           TBEN_L4_8IOL:I.Data[155].0   // IO-Link event 8 - Qualifier (INT bit0)
           TBEN_L4_8IOL:I.Data[155].1   // IO-Link event 8 - Qualifier (INT bit1)
           TBEN_L4_8IOL:I.Data[155].10   // IO-Link event 8 - Port (INT bit2)
           TBEN_L4_8IOL:I.Data[155].11   // IO-Link event 8 - Port (INT bit3)
           TBEN_L4_8IOL:I.Data[155].12   // IO-Link event 8 - Port (INT bit4)
           TBEN_L4_8IOL:I.Data[155].13   // IO-Link event 8 - Port (INT bit5)
           TBEN_L4_8IOL:I.Data[155].14   // IO-Link event 8 - Port (INT bit6)
           TBEN_L4_8IOL:I.Data[155].15   // IO-Link event 8 - Port (INT bit7)
           TBEN_L4_8IOL:I.Data[155].2   // IO-Link event 8 - Qualifier (INT bit2)
           TBEN_L4_8IOL:I.Data[155].3   // IO-Link event 8 - Qualifier (INT bit3)
           TBEN_L4_8IOL:I.Data[155].4   // IO-Link event 8 - Qualifier (INT bit4)
           TBEN_L4_8IOL:I.Data[155].5   // IO-Link event 8 - Qualifier (INT bit5)
           TBEN_L4_8IOL:I.Data[155].6   // IO-Link event 8 - Qualifier (INT bit6)
           TBEN_L4_8IOL:I.Data[155].7   // IO-Link event 8 - Qualifier (INT bit7)
           TBEN_L4_8IOL:I.Data[155].8   // IO-Link event 8 - Port (INT bit0)
           TBEN_L4_8IOL:I.Data[155].9   // IO-Link event 8 - Port (INT bit1)
           TBEN_L4_8IOL:I.Data[156]   // IO-Link event 8 - Event code
           TBEN_L4_8IOL:I.Data[156].0   // IO-Link event 8 - Event code (INT bit0)
           TBEN_L4_8IOL:I.Data[156].1   // IO-Link event 8 - Event code (INT bit1)
           TBEN_L4_8IOL:I.Data[156].10   // IO-Link event 8 - Event code (INT bit10)
           TBEN_L4_8IOL:I.Data[156].11   // IO-Link event 8 - Event code (INT bit11)
           TBEN_L4_8IOL:I.Data[156].12   // IO-Link event 8 - Event code (INT bit12)
           TBEN_L4_8IOL:I.Data[156].13   // IO-Link event 8 - Event code (INT bit13)
           TBEN_L4_8IOL:I.Data[156].14   // IO-Link event 8 - Event code (INT bit14)
           TBEN_L4_8IOL:I.Data[156].15   // IO-Link event 8 - Event code (INT bit15)
           TBEN_L4_8IOL:I.Data[156].2   // IO-Link event 8 - Event code (INT bit2)
           TBEN_L4_8IOL:I.Data[156].3   // IO-Link event 8 - Event code (INT bit3)
           TBEN_L4_8IOL:I.Data[156].4   // IO-Link event 8 - Event code (INT bit4)
           TBEN_L4_8IOL:I.Data[156].5   // IO-Link event 8 - Event code (INT bit5)
           TBEN_L4_8IOL:I.Data[156].6   // IO-Link event 8 - Event code (INT bit6)
           TBEN_L4_8IOL:I.Data[156].7   // IO-Link event 8 - Event code (INT bit7)
           TBEN_L4_8IOL:I.Data[156].8   // IO-Link event 8 - Event code (INT bit8)
           TBEN_L4_8IOL:I.Data[156].9   // IO-Link event 8 - Event code (INT bit9)
           TBEN_L4_8IOL:I.Data[157]   // IO-Link event 9 - Qualifier, IO-Link event 9 - Port
           TBEN_L4_8IOL:I.Data[157].0   // IO-Link event 9 - Qualifier (INT bit0)
           TBEN_L4_8IOL:I.Data[157].1   // IO-Link event 9 - Qualifier (INT bit1)
           TBEN_L4_8IOL:I.Data[157].10   // IO-Link event 9 - Port (INT bit2)
           TBEN_L4_8IOL:I.Data[157].11   // IO-Link event 9 - Port (INT bit3)
           TBEN_L4_8IOL:I.Data[157].12   // IO-Link event 9 - Port (INT bit4)
           TBEN_L4_8IOL:I.Data[157].13   // IO-Link event 9 - Port (INT bit5)
           TBEN_L4_8IOL:I.Data[157].14   // IO-Link event 9 - Port (INT bit6)
           TBEN_L4_8IOL:I.Data[157].15   // IO-Link event 9 - Port (INT bit7)
           TBEN_L4_8IOL:I.Data[157].2   // IO-Link event 9 - Qualifier (INT bit2)
           TBEN_L4_8IOL:I.Data[157].3   // IO-Link event 9 - Qualifier (INT bit3)
           TBEN_L4_8IOL:I.Data[157].4   // IO-Link event 9 - Qualifier (INT bit4)
           TBEN_L4_8IOL:I.Data[157].5   // IO-Link event 9 - Qualifier (INT bit5)
           TBEN_L4_8IOL:I.Data[157].6   // IO-Link event 9 - Qualifier (INT bit6)
           TBEN_L4_8IOL:I.Data[157].7   // IO-Link event 9 - Qualifier (INT bit7)
           TBEN_L4_8IOL:I.Data[157].8   // IO-Link event 9 - Port (INT bit0)
